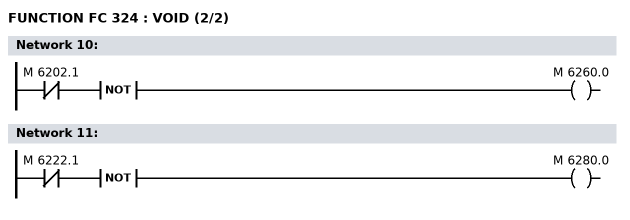

      AN    M   6202.1;
      NOT   ;
      =     M   6260.0;
NETWORK
TITLE =

      AN    M   6222.1;
      NOT   ;
      =     M   6280.0;
END_FUNCTION

FUNCTION_BLOCK FB 406
TITLE =Data Block Move Program
AUTHOR : HMC
FAMILY : Car_Type
NAME : Car_Type
VERSION : 1.0


VAR_INPUT
  FWD_Pulse : BOOL ;
  RET_Pulse : BOOL ;
  Source_DB : INT ;
  Start_Add : INT ;
  Stn_Amount : INT ;
  Byte_per_Stn : INT ;
  Cpu_Run_Pulse : BOOL ;
END_VAR
VAR_OUTPUT
  Complete : BOOL ;
END_VAR
VAR
  Operation : BOOL ;
  Mask_Arr : ARRAY  [0 .. 599 ] OF BYTE ;
  Ret : INT ;
  Data_Type : WORD ;
  Data_Length : INT ;
  Secend_Stn_Add : INT ;
  Fill_Source : WORD ;
END_VAR
VAR_TEMP
  First_Stn : ANY ;
  Mask : ANY ;
  Second_Stn : ANY ;
  Save_AR1 : DWORD ;
  Save_AR2 : DWORD ;
  Save_DB : INT ;
  Save_DI : INT ;
  First_Stn_1 : ANY ;
END_VAR
BEGIN
NETWORK
TITLE =Save adress register and DB's

      TAR1  #Save_AR1; // Save adress register 1
      TAR2  #Save_AR2; // Save adress register 2
      L     DBNO; // loads the number of the shared open data block
      T     #Save_DB;
      L     DINO; // loads the number of the opened instance data block
      T     #Save_DI;
NETWORK
TITLE =Operation Pulse

      O     #FWD_Pulse; // External ForwardOperation Signal
      O     #RET_Pulse; // External Return Operation Signal
      FP    #Operation; // Operation Pulse
      JNB   _End; // Jump to End
NETWORK
TITLE =Data Type Select In ANY Type Parameter

      A(    ; // If Source DB is Not Zero
      L     #Source_DB;
      L     0;
      <>I   ;
      )     ;
      JNB   _001; // Jump to Next Step
      L     W#16#8400; // Load "8400" _ Means "DB Area"
      T     #Data_Type; // Transfer to Data_Type
_001: NOP   0;
NETWORK
TITLE =Data Type Select In ANY Type Parameter

      A(    ; // If DB_NO is Zero
      L     #Source_DB;
      L     0;
      ==I   ;
      )     ;
      JNB   _002; // Jump to Next Step
      L     W#16#8300; // Load "8300" _ Means "Bit Memory Area"
      T     #Data_Type; // Transfer to Data_Type
_002: NOP   0;
NETWORK
TITLE =Data Length Select

      L     #Stn_Amount; // Station Amount - 1
      L     1;
      -I    ;
      L     #Byte_per_Stn; // Multi Length Per Station
      *I    ;
      T     #Data_Length; // Transfer to Data Length
NETWORK
TITLE =2nd Station Address Select

      L     #Start_Add; // Pluse Start Address And Length
      L     #Byte_per_Stn;
      +I    ;
      T     #Secend_Stn_Add; // Transfer to Second Station Address
NETWORK
TITLE =Make a "ANY" Type Data

      LAR1  P##First_Stn; // Load 1st Station Address of ANY Pointer In "AR1"

      L     B#16#10; // Load Syntax ID For S7 "10"
      T     LB [AR1,P#0.0]; // Transfer ID to the ANY Pointer

      L     B#16#2; // Load Data Type _ "2" means "BYTE"
      T     LB [AR1,P#1.0]; // Transfer Data Type to the ANY Pointer

      L     #Data_Length; // Load the Length of Source Data
      T     LW [AR1,P#2.0]; // Transfer the Numbers to the ANY Pointer

      L     #Source_DB; // Load DB Number _ "0" means don't use "DB"
      T     LW [AR1,P#4.0]; // Transfer the Numbers to the ANY Pointer

      L     #Data_Type; // Load Data Type _ "83" means "Bit Memory" Area
      T     LW [AR1,P#6.0]; //                  "84" means "DB" Area

      L     #Start_Add; // Load Start Address
      SLW   3; // Shift Left Word _ "3" Bit
      T     LW [AR1,P#8.0]; // Transfer the Address to the ANY Pointer

      LAR1  P##Mask; // Load 2nd Station Address of ANY Pointer In "AR1"

      L     B#16#10; //Load Syntax ID For S7 "10"
      T     LB [AR1,P#0.0]; //Load Syntax ID For S7 "10"

      L     B#16#2; //  Load Data Type _ "2" means "BYTE"
      T     LB [AR1,P#1.0]; // Transfer Data Type to the ANY Pointer

      L     #Data_Length; // Load the Length of Target Data
      T     LW [AR1,P#2.0]; // Transfer the Numbers to the ANY Pointer

      L     #Save_DI; // Load DB Number _ "0" means don't use "DB"
      T     LW [AR1,P#4.0]; // Transfer the Numbers to the ANY Pointer

      L     #Data_Type; // Load Data Type _ "83" means "Bit Memory" Area
      T     LW [AR1,P#6.0]; //                  "84" means "DB" Area

      L     16; //  Load Start Address
      SLW   3; // Shift Left Word _ "3" Bit
      T     LW [AR1,P#8.0]; // Transfer the Address to the ANY Pointer

NETWORK
TITLE =Make a "ANY" Type Data

      LAR1  P##Second_Stn; // Load 1st Station Address of ANY Pointer In "AR1"

      L     B#16#10; // Load Syntax ID For S7 "10"
      T     LB [AR1,P#0.0]; // Transfer ID to the ANY Pointer

      L     B#16#2; // Load Data Type _ "2" means "BYTE"
      T     LB [AR1,P#1.0]; // Transfer Data Type to the ANY Pointer

      L     #Data_Length; // Load the Length of Source Data
      T     LW [AR1,P#2.0]; // Transfer the Numbers to the ANY Pointer

      L     #Source_DB; // Load DB Number _ "0" means don't use "DB"
      T     LW [AR1,P#4.0]; // Transfer the Numbers to the ANY Pointer

      L     #Data_Type; // Load Data Type _ "83" means "Bit Memory" Area
      T     LW [AR1,P#6.0]; //                  "84" means "DB" Area

      L     #Secend_Stn_Add; // Load Second Station Address
      SLW   3; // Shift Left Word _ "3" Bit
      T     LW [AR1,P#8.0]; // Transfer the Address to the ANY Pointer
NETWORK
TITLE =Reset Car Type Transfer Complete Signal

      O     #FWD_Pulse; // External Forward Operation Signal
      O     #RET_Pulse; // External Return Operation Signal
      R     #Complete; // Reset Complete Signal
NETWORK
TITLE =Make Fill Source Data

      L     0;
      T     #Fill_Source;
NETWORK
TITLE =Fwd Block Move to Mask Area

      A     #FWD_Pulse; // External Forward Operation Signal
      AN    #Complete; // Complete Signal is False
      AN    #Cpu_Run_Pulse;
      JNB   _FWD;
      CALL SFC   20 (
           SRCBLK                   := #First_Stn,
           RET_VAL                  := #Ret,
           DSTBLK                   := #Mask);

NETWORK
TITLE =Clear Source Data Area


      CALL SFC   21 (
           BVAL                     := #Fill_Source,// "Zero"
           RET_VAL                  := #Ret,
           BLK                      := #First_Stn);// Transfer to First Station Area

NETWORK
TITLE =Fwd Block Move to Second Station Area


      CALL SFC   20 (
           SRCBLK                   := #Mask,
           RET_VAL                  := #Ret,
           DSTBLK                   := #Second_Stn);

NETWORK
TITLE =Clear Mask Data Area


      CALL SFC   21 (
           BVAL                     := #Fill_Source,// "Zero"
           RET_VAL                  := #Ret,
           BLK                      := #Mask);// Transfer to Mask Area
_FWD: NOP   0;
NETWORK
TITLE =Rev Block Move to Mask Area

      A     #RET_Pulse; // External Return Operation Signal
      AN    #Complete; // Complete Signal is False
      AN    #Cpu_Run_Pulse;
      JNB   _REV;
      CALL SFC   20 (
           SRCBLK                   := #Second_Stn,
           RET_VAL                  := #Ret,
           DSTBLK                   := #Mask);

NETWORK
TITLE =Clear Source Data Area


      CALL SFC   21 (
           BVAL                     := #Fill_Source,// "Zero"
           RET_VAL                  := #Ret,
           BLK                      := #Second_Stn);// Transfer to Second Station Area

NETWORK
TITLE =Rev Block Move to First Station Area


      CALL SFC   20 (
           SRCBLK                   := #Mask,
           RET_VAL                  := #Ret,
           DSTBLK                   := #First_Stn);

NETWORK
TITLE =Clear Mask Data Area


      CALL SFC   21 (
           BVAL                     := #Fill_Source,// "Zero"
           RET_VAL                  := #Ret,
           BLK                      := #Mask);// Transfer to Mask Area
_REV: NOP   0;
NETWORK
TITLE =Set Complete Signal

      S     #Complete;
_End: NOP   0;
END_FUNCTION_BLOCK

FUNCTION_BLOCK FB 426
TITLE =Sensor Error,Lamp Variables Program
AUTHOR : HMC
FAMILY : Common
NAME : Common
VERSION : 1.0


VAR_INPUT
  Enable_Aux : BOOL ;
  Adv_Amount : INT ;
  Ret_Amount : INT ;
  LS_Adv1 : BOOL ;
  LS_Ret1 : BOOL ;
  LS_Adv2 : BOOL ;
  LS_Ret2 : BOOL ;
  LS_Adv3 : BOOL ;
  LS_Ret3 : BOOL ;
  LS_Adv4 : BOOL ;
  LS_Ret4 : BOOL ;
  LS_Adv5 : BOOL ;
  LS_Ret5 : BOOL ;
  LS_Adv6 : BOOL ;
  LS_Ret6 : BOOL ;
  LS_Adv7 : BOOL ;
  LS_Ret7 : BOOL ;
  LS_Adv8 : BOOL ;
  LS_Ret8 : BOOL ;
  SOL_Adv : BOOL ;
  SOL_Ret : BOOL ;
  M_Ready : BOOL ;
  T_CHK1 : TIME ;
  T_CHK2 : TIME ;
  PB_Lamp_CHK : BOOL ;
  PB_Error_Rst : BOOL ;
  M_FLICK : BOOL ;
END_VAR
VAR_OUTPUT
  M_Adv_Err : BOOL ;
  M_Ret_Err : BOOL ;
  LP_Adv : BOOL ;
  LP_Ret : BOOL ;
  Visu_Adv : WORD ;
  Visu_Ret : WORD ;
END_VAR
VAR
  Error_T1 : SFB 4;
  Error_T2 : SFB 4;
  Adv_End_Aux : BOOL ;
  Ret_End_Aux : BOOL ;
  CHK_Aux1 : BOOL ;
  CHK_Aux2 : BOOL ;
  Error_T1_DN : BOOL ;
  Error_T2_DN : BOOL ;
  Adv_Memo : BOOL ;
  Visu_Adv_Arr : ARRAY  [0 .. 15 ] OF BOOL ;
  Visu_Ret_Arr : ARRAY  [0 .. 15 ] OF BOOL ;
  BLK_Move_Ret : INT ;
  Enable : BOOL ;
  Adv_End : BOOL ;
  Ret_End : BOOL ;
END_VAR
BEGIN
NETWORK
TITLE =
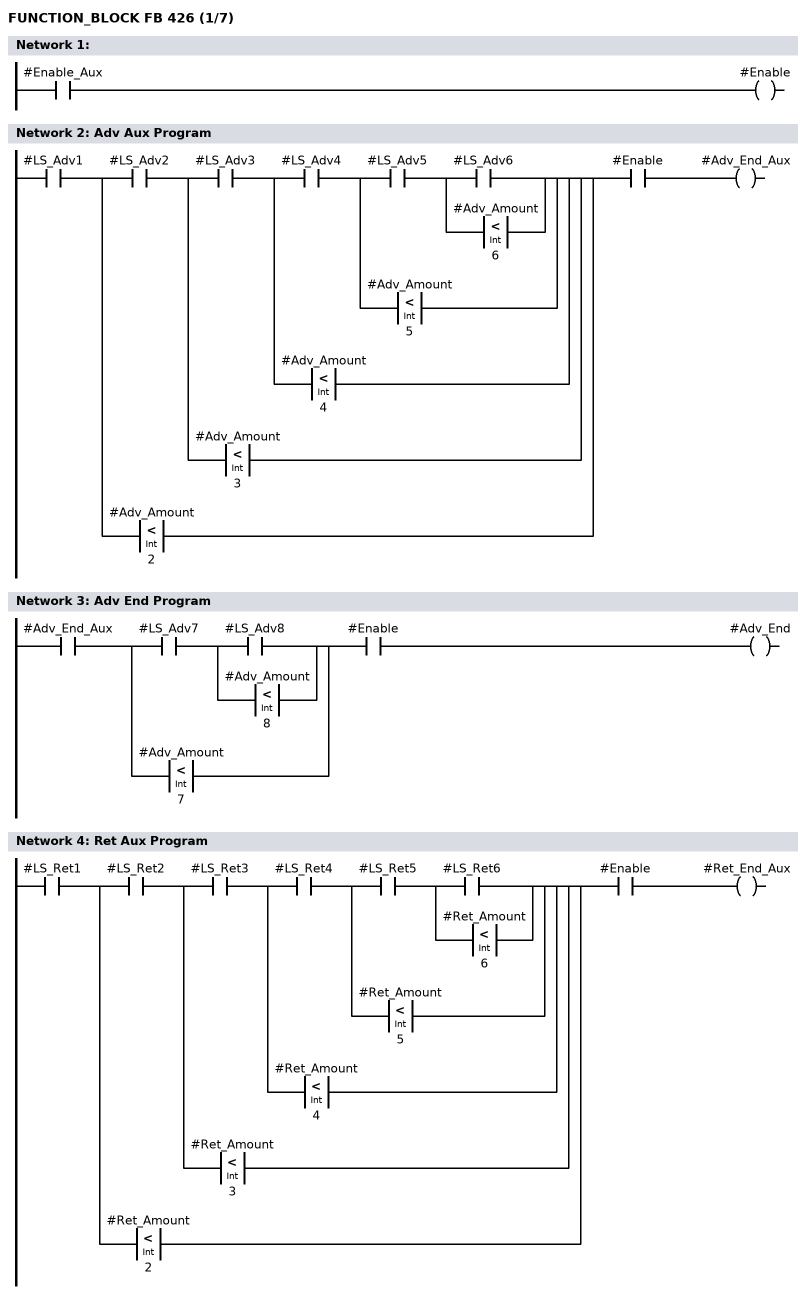

      A     #Enable_Aux;
      =     #Enable;
NETWORK
TITLE =Adv Aux Program

      A     #LS_Adv1;
      A(    ;
      A     #LS_Adv2;
      A(    ;
      A     #LS_Adv3;
      A(    ;
      A     #LS_Adv4;
      A(    ;
      A     #LS_Adv5;
      A(    ;
      O     #LS_Adv6;
      O(    ;
      L     #Adv_Amount;
      L     6;
      <I    ;
      )     ;
      )     ;
      O(    ;
      L     #Adv_Amount;
      L     5;
      <I    ;
      )     ;
      )     ;
      O(    ;
      L     #Adv_Amount;
      L     4;
      <I    ;
      )     ;
      )     ;
      O(    ;
      L     #Adv_Amount;
      L     3;
      <I    ;
      )     ;
      )     ;
      O(    ;
      L     #Adv_Amount;
      L     2;
      <I    ;
      )     ;
      )     ;
      A     #Enable;
      =     #Adv_End_Aux;
NETWORK
TITLE =Adv End Program

      A     #Adv_End_Aux;
      A(    ;
      A     #LS_Adv7;
      A(    ;
      O     #LS_Adv8;
      O(    ;
      L     #Adv_Amount;
      L     8;
      <I    ;
      )     ;
      )     ;
      O(    ;
      L     #Adv_Amount;
      L     7;
      <I    ;
      )     ;
      )     ;
      A     #Enable;
      =     #Adv_End;
NETWORK
TITLE =Ret Aux Program

      A     #LS_Ret1;
      A(    ;
      A     #LS_Ret2;
      A(    ;
      A     #LS_Ret3;
      A(    ;
      A     #LS_Ret4;
      A(    ;
      A     #LS_Ret5;
      A(    ;
      O     #LS_Ret6;
      O(    ;
      L     #Ret_Amount;
      L     6;
      <I    ;
      )     ;
      )     ;
      O(    ;
      L     #Ret_Amount;
      L     5;
      <I    ;
      )     ;
      )     ;
      O(    ;
      L     #Ret_Amount;
      L     4;
      <I    ;
      )     ;
      )     ;
      O(    ;
      L     #Ret_Amount;
      L     3;
      <I    ;
      )     ;
      )     ;
      O(    ;
      L     #Ret_Amount;
      L     2;
      <I    ;
      )     ;
      )     ;
      A     #Enable;
      =     #Ret_End_Aux;
NETWORK
TITLE =Ret End Program
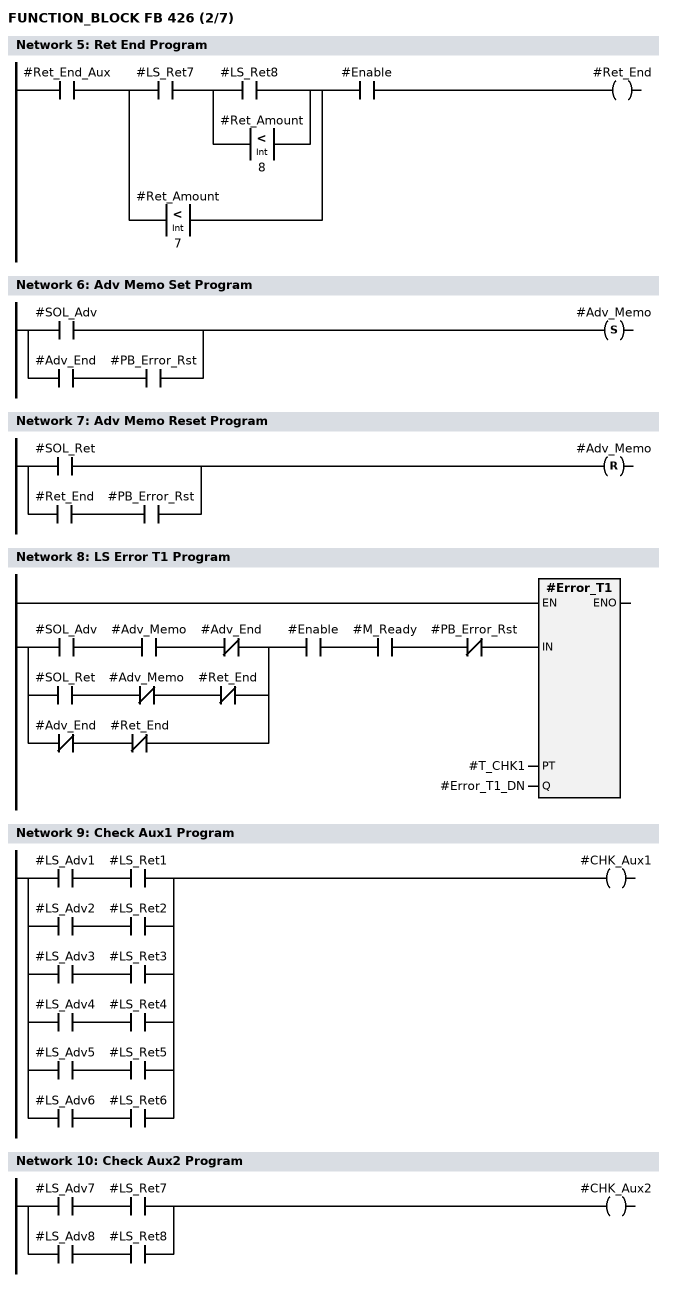

      A     #Ret_End_Aux;
      A(    ;
      A     #LS_Ret7;
      A(    ;
      O     #LS_Ret8;
      O(    ;
      L     #Ret_Amount;
      L     8;
      <I    ;
      )     ;
      )     ;
      O(    ;
      L     #Ret_Amount;
      L     7;
      <I    ;
      )     ;
      )     ;
      A     #Enable;
      =     #Ret_End;
NETWORK
TITLE =Adv Memo Set Program

      O     #SOL_Adv;
      O     ;
      A     #Adv_End;
      A     #PB_Error_Rst;
      S     #Adv_Memo;
NETWORK
TITLE =Adv Memo Reset Program

      O     #SOL_Ret;
      O     ;
      A     #Ret_End;
      A     #PB_Error_Rst;
      R     #Adv_Memo;
NETWORK
TITLE =LS Error T1 Program

      A(    ;
      A     #SOL_Adv;
      A     #Adv_Memo;
      AN    #Adv_End;
      O     ;
      A     #SOL_Ret;
      AN    #Adv_Memo;
      AN    #Ret_End;
      O     ;
      AN    #Adv_End;
      AN    #Ret_End;
      )     ;
      A     #Enable;
      A     #M_Ready;
      AN    #PB_Error_Rst;
      =     L      0.0;
      BLD   103;
      CALL #Error_T1 (
           IN                       := L      0.0,
           PT                       := #T_CHK1,
           Q                        := #Error_T1_DN);

      NOP   0;
NETWORK
TITLE =Check Aux1 Program

      A     #LS_Adv1;
      A     #LS_Ret1;
      O     ;
      A     #LS_Adv2;
      A     #LS_Ret2;
      O     ;
      A     #LS_Adv3;
      A     #LS_Ret3;
      O     ;
      A     #LS_Adv4;
      A     #LS_Ret4;
      O     ;
      A     #LS_Adv5;
      A     #LS_Ret5;
      O     ;
      A     #LS_Adv6;
      A     #LS_Ret6;
      =     #CHK_Aux1;
NETWORK
TITLE =Check Aux2 Program

      A     #LS_Adv7;
      A     #LS_Ret7;
      O     ;
      A     #LS_Adv8;
      A     #LS_Ret8;
      =     #CHK_Aux2;
NETWORK
TITLE =LS Error T2 Program
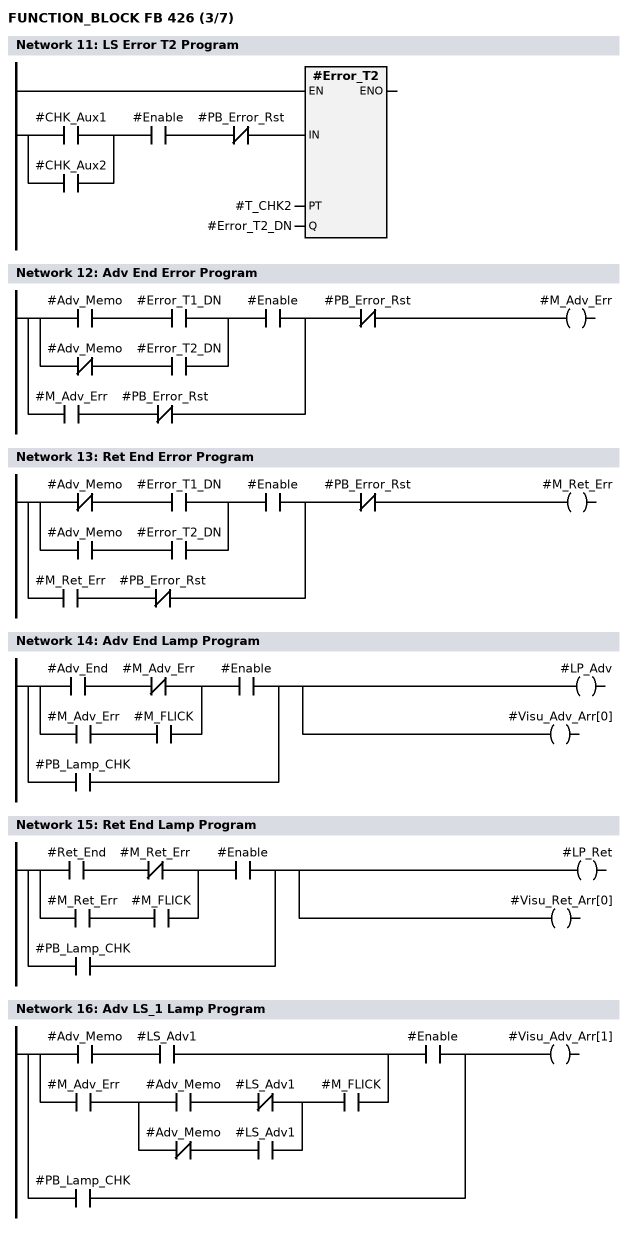

      A(    ;
      O     #CHK_Aux1;
      O     #CHK_Aux2;
      )     ;
      A     #Enable;
      AN    #PB_Error_Rst;
      =     L      0.0;
      BLD   103;
      CALL #Error_T2 (
           IN                       := L      0.0,
           PT                       := #T_CHK2,
           Q                        := #Error_T2_DN);

      NOP   0;
NETWORK
TITLE =Adv End Error Program

      A(    ;
      A(    ;
      A     #Adv_Memo;
      A     #Error_T1_DN;
      O     ;
      AN    #Adv_Memo;
      A     #Error_T2_DN;
      )     ;
      A     #Enable;
      O     ;
      A     #M_Adv_Err;
      AN    #PB_Error_Rst;
      )     ;
      AN    #PB_Error_Rst;
      =     #M_Adv_Err;
NETWORK
TITLE =Ret End Error Program

      A(    ;
      A(    ;
      AN    #Adv_Memo;
      A     #Error_T1_DN;
      O     ;
      A     #Adv_Memo;
      A     #Error_T2_DN;
      )     ;
      A     #Enable;
      O     ;
      A     #M_Ret_Err;
      AN    #PB_Error_Rst;
      )     ;
      AN    #PB_Error_Rst;
      =     #M_Ret_Err;
NETWORK
TITLE =Adv End Lamp Program

      A(    ;
      A     #Adv_End;
      AN    #M_Adv_Err;
      O     ;
      A     #M_Adv_Err;
      A     #M_FLICK;
      )     ;
      A     #Enable;
      O     #PB_Lamp_CHK;
      =     #LP_Adv;
      =     #Visu_Adv_Arr[0];
NETWORK
TITLE =Ret End Lamp Program

      A(    ;
      A     #Ret_End;
      AN    #M_Ret_Err;
      O     ;
      A     #M_Ret_Err;
      A     #M_FLICK;
      )     ;
      A     #Enable;
      O     #PB_Lamp_CHK;
      =     #LP_Ret;
      =     #Visu_Ret_Arr[0];
NETWORK
TITLE =Adv LS_1 Lamp Program

      A(    ;
      A     #Adv_Memo;
      A     #LS_Adv1;
      O     ;
      A     #M_Adv_Err;
      A(    ;
      A     #Adv_Memo;
      AN    #LS_Adv1;
      O     ;
      AN    #Adv_Memo;
      A     #LS_Adv1;
      )     ;
      A     #M_FLICK;
      )     ;
      A     #Enable;
      O     #PB_Lamp_CHK;
      =     #Visu_Adv_Arr[1];
NETWORK
TITLE =Adv LS_2 Lamp Program
//
//
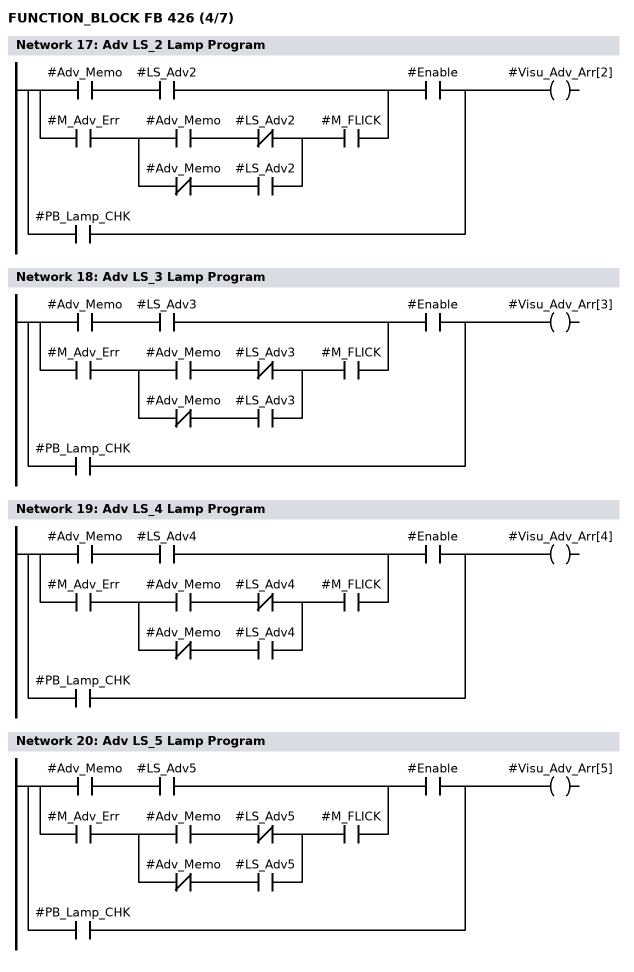
      A(    ;
      A     #Adv_Memo;
      A     #LS_Adv2;
      O     ;
      A     #M_Adv_Err;
      A(    ;
      A     #Adv_Memo;
      AN    #LS_Adv2;
      O     ;
      AN    #Adv_Memo;
      A     #LS_Adv2;
      )     ;
      A     #M_FLICK;
      )     ;
      A     #Enable;
      O     #PB_Lamp_CHK;
      =     #Visu_Adv_Arr[2];
NETWORK
TITLE =Adv LS_3 Lamp Program
//
//
      A(    ;
      A     #Adv_Memo;
      A     #LS_Adv3;
      O     ;
      A     #M_Adv_Err;
      A(    ;
      A     #Adv_Memo;
      AN    #LS_Adv3;
      O     ;
      AN    #Adv_Memo;
      A     #LS_Adv3;
      )     ;
      A     #M_FLICK;
      )     ;
      A     #Enable;
      O     #PB_Lamp_CHK;
      =     #Visu_Adv_Arr[3];
NETWORK
TITLE =Adv LS_4 Lamp Program
//
//
      A(    ;
      A     #Adv_Memo;
      A     #LS_Adv4;
      O     ;
      A     #M_Adv_Err;
      A(    ;
      A     #Adv_Memo;
      AN    #LS_Adv4;
      O     ;
      AN    #Adv_Memo;
      A     #LS_Adv4;
      )     ;
      A     #M_FLICK;
      )     ;
      A     #Enable;
      O     #PB_Lamp_CHK;
      =     #Visu_Adv_Arr[4];
NETWORK
TITLE =Adv LS_5 Lamp Program
//
//
      A(    ;
      A     #Adv_Memo;
      A     #LS_Adv5;
      O     ;
      A     #M_Adv_Err;
      A(    ;
      A     #Adv_Memo;
      AN    #LS_Adv5;
      O     ;
      AN    #Adv_Memo;
      A     #LS_Adv5;
      )     ;
      A     #M_FLICK;
      )     ;
      A     #Enable;
      O     #PB_Lamp_CHK;
      =     #Visu_Adv_Arr[5];
NETWORK
TITLE =Adv LS_6 Lamp Program
//
//
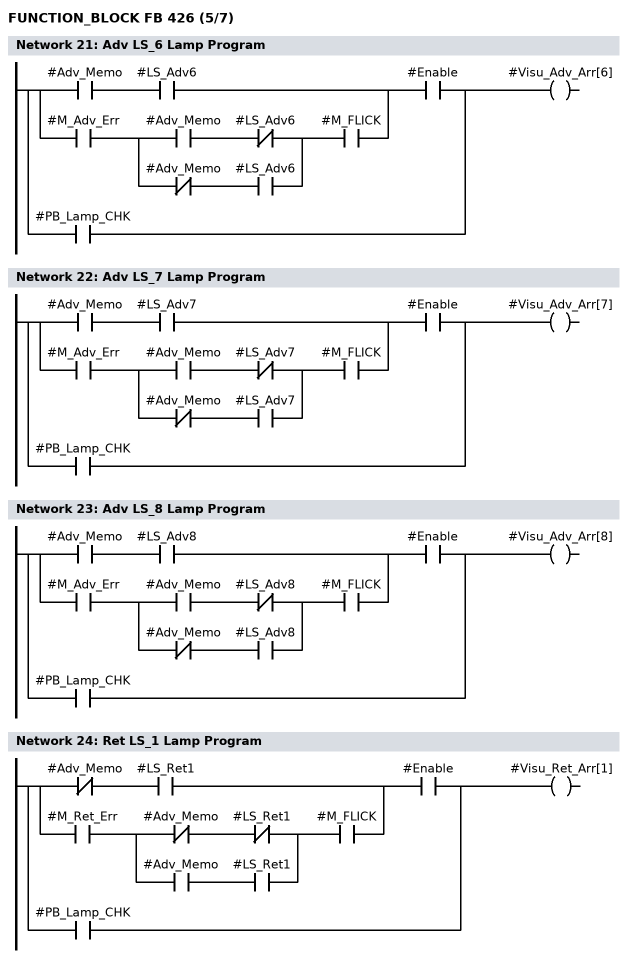
      A(    ;
      A     #Adv_Memo;
      A     #LS_Adv6;
      O     ;
      A     #M_Adv_Err;
      A(    ;
      A     #Adv_Memo;
      AN    #LS_Adv6;
      O     ;
      AN    #Adv_Memo;
      A     #LS_Adv6;
      )     ;
      A     #M_FLICK;
      )     ;
      A     #Enable;
      O     #PB_Lamp_CHK;
      =     #Visu_Adv_Arr[6];
NETWORK
TITLE =Adv LS_7 Lamp Program
//
//
      A(    ;
      A     #Adv_Memo;
      A     #LS_Adv7;
      O     ;
      A     #M_Adv_Err;
      A(    ;
      A     #Adv_Memo;
      AN    #LS_Adv7;
      O     ;
      AN    #Adv_Memo;
      A     #LS_Adv7;
      )     ;
      A     #M_FLICK;
      )     ;
      A     #Enable;
      O     #PB_Lamp_CHK;
      =     #Visu_Adv_Arr[7];
NETWORK
TITLE =Adv LS_8 Lamp Program
//
//
      A(    ;
      A     #Adv_Memo;
      A     #LS_Adv8;
      O     ;
      A     #M_Adv_Err;
      A(    ;
      A     #Adv_Memo;
      AN    #LS_Adv8;
      O     ;
      AN    #Adv_Memo;
      A     #LS_Adv8;
      )     ;
      A     #M_FLICK;
      )     ;
      A     #Enable;
      O     #PB_Lamp_CHK;
      =     #Visu_Adv_Arr[8];
NETWORK
TITLE =Ret LS_1 Lamp Program
//
//
      A(    ;
      AN    #Adv_Memo;
      A     #LS_Ret1;
      O     ;
      A     #M_Ret_Err;
      A(    ;
      AN    #Adv_Memo;
      AN    #LS_Ret1;
      O     ;
      A     #Adv_Memo;
      A     #LS_Ret1;
      )     ;
      A     #M_FLICK;
      )     ;
      A     #Enable;
      O     #PB_Lamp_CHK;
      =     #Visu_Ret_Arr[1];
NETWORK
TITLE =Ret LS_2 Lamp Program
//
//
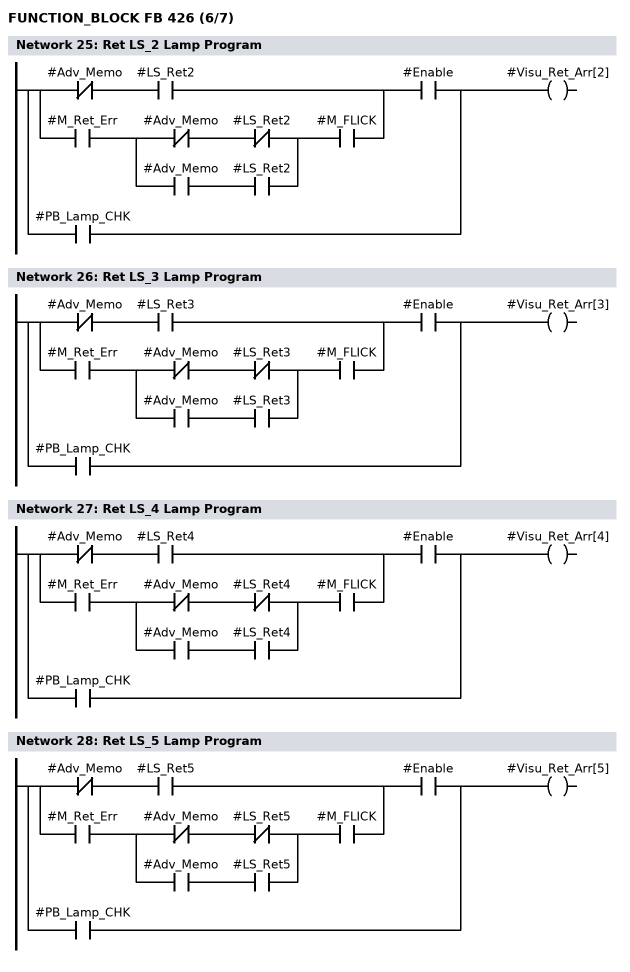
      A(    ;
      AN    #Adv_Memo;
      A     #LS_Ret2;
      O     ;
      A     #M_Ret_Err;
      A(    ;
      AN    #Adv_Memo;
      AN    #LS_Ret2;
      O     ;
      A     #Adv_Memo;
      A     #LS_Ret2;
      )     ;
      A     #M_FLICK;
      )     ;
      A     #Enable;
      O     #PB_Lamp_CHK;
      =     #Visu_Ret_Arr[2];
NETWORK
TITLE =Ret LS_3 Lamp Program
//
//
      A(    ;
      AN    #Adv_Memo;
      A     #LS_Ret3;
      O     ;
      A     #M_Ret_Err;
      A(    ;
      AN    #Adv_Memo;
      AN    #LS_Ret3;
      O     ;
      A     #Adv_Memo;
      A     #LS_Ret3;
      )     ;
      A     #M_FLICK;
      )     ;
      A     #Enable;
      O     #PB_Lamp_CHK;
      =     #Visu_Ret_Arr[3];
NETWORK
TITLE =Ret LS_4 Lamp Program
//
//
      A(    ;
      AN    #Adv_Memo;
      A     #LS_Ret4;
      O     ;
      A     #M_Ret_Err;
      A(    ;
      AN    #Adv_Memo;
      AN    #LS_Ret4;
      O     ;
      A     #Adv_Memo;
      A     #LS_Ret4;
      )     ;
      A     #M_FLICK;
      )     ;
      A     #Enable;
      O     #PB_Lamp_CHK;
      =     #Visu_Ret_Arr[4];
NETWORK
TITLE =Ret LS_5 Lamp Program
//
//
      A(    ;
      AN    #Adv_Memo;
      A     #LS_Ret5;
      O     ;
      A     #M_Ret_Err;
      A(    ;
      AN    #Adv_Memo;
      AN    #LS_Ret5;
      O     ;
      A     #Adv_Memo;
      A     #LS_Ret5;
      )     ;
      A     #M_FLICK;
      )     ;
      A     #Enable;
      O     #PB_Lamp_CHK;
      =     #Visu_Ret_Arr[5];
NETWORK
TITLE =Ret LS_6 Lamp Program
//
//
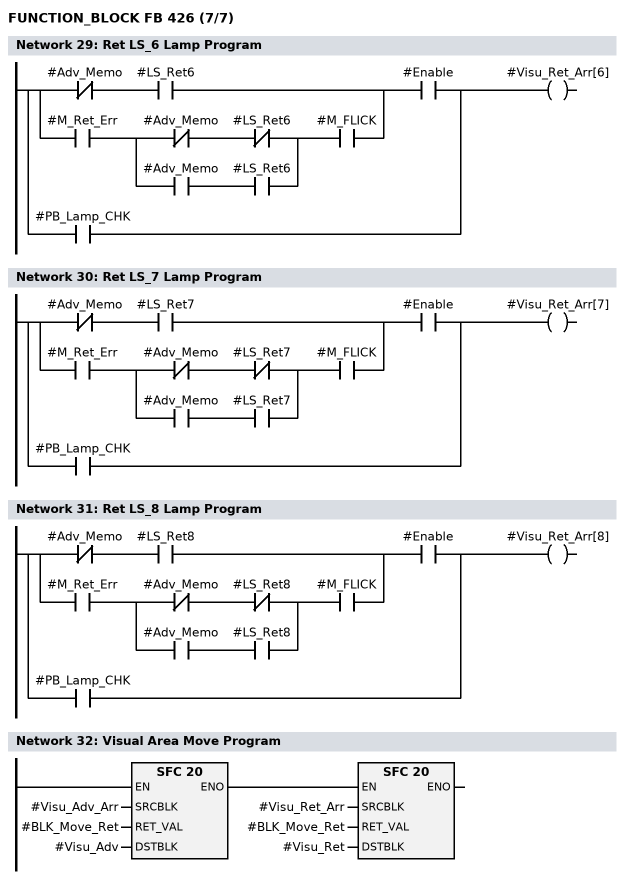
      A(    ;
      AN    #Adv_Memo;
      A     #LS_Ret6;
      O     ;
      A     #M_Ret_Err;
      A(    ;
      AN    #Adv_Memo;
      AN    #LS_Ret6;
      O     ;
      A     #Adv_Memo;
      A     #LS_Ret6;
      )     ;
      A     #M_FLICK;
      )     ;
      A     #Enable;
      O     #PB_Lamp_CHK;
      =     #Visu_Ret_Arr[6];
NETWORK
TITLE =Ret LS_7 Lamp Program
//
//
      A(    ;
      AN    #Adv_Memo;
      A     #LS_Ret7;
      O     ;
      A     #M_Ret_Err;
      A(    ;
      AN    #Adv_Memo;
      AN    #LS_Ret7;
      O     ;
      A     #Adv_Memo;
      A     #LS_Ret7;
      )     ;
      A     #M_FLICK;
      )     ;
      A     #Enable;
      O     #PB_Lamp_CHK;
      =     #Visu_Ret_Arr[7];
NETWORK
TITLE =Ret LS_8 Lamp Program
//
//
      A(    ;
      AN    #Adv_Memo;
      A     #LS_Ret8;
      O     ;
      A     #M_Ret_Err;
      A(    ;
      AN    #Adv_Memo;
      AN    #LS_Ret8;
      O     ;
      A     #Adv_Memo;
      A     #LS_Ret8;
      )     ;
      A     #M_FLICK;
      )     ;
      A     #Enable;
      O     #PB_Lamp_CHK;
      =     #Visu_Ret_Arr[8];
NETWORK
TITLE =Visual Area Move Program

      A(    ;
      CALL SFC   20 (
           SRCBLK                   := #Visu_Adv_Arr,
           RET_VAL                  := #BLK_Move_Ret,
           DSTBLK                   := #Visu_Adv);
      A     BR;
      )     ;
      JNB   _001;
      CALL SFC   20 (
           SRCBLK                   := #Visu_Ret_Arr,
           RET_VAL                  := #BLK_Move_Ret,
           DSTBLK                   := #Visu_Ret);
_001: NOP   0;
END_FUNCTION_BLOCK

FUNCTION_BLOCK FB 475
TITLE =ProfiBus DP Communication Fault Variables Program
AUTHOR : HMC
FAMILY : Drive
NAME : Drive
VERSION : 1.0


VAR_INPUT
  M_Check_Active : BOOL ;
  DP_Not_Pre_Byte : BYTE ;	//Startadress Outputs from HW-Konfig
  DP_Error_Byte : BYTE ;	//Startadress Inputs from HW-Konfig
  M_Error_Rst : BOOL ;
END_VAR
VAR_OUTPUT
  Node0_Fault : BOOL ;
  Node1_Fault : BOOL ;
  Node2_Fault : BOOL ;
  Node3_Fault : BOOL ;
  Node4_Fault : BOOL ;
  Node5_Fault : BOOL ;
  Node6_Fault : BOOL ;
  Node7_Fault : BOOL ;
END_VAR
VAR
  Pre_Arr : ARRAY  [0 .. 7 ] OF BOOL ;
  Fault_Arr : ARRAY  [0 .. 7 ] OF BOOL ;
  node_0_err : SFB 4;
  node_1_err : SFB 4;
  node_2_err : SFB 4;
  node_3_err : SFB 4;
  node_4_err : SFB 4;
  node_5_err : SFB 4;
  node_6_err : SFB 4;
  node_7_err : SFB 4;
END_VAR
VAR_TEMP
  Ret : INT ;
END_VAR
BEGIN
NETWORK
TITLE =DP Fault Byte Move To DP Fault Array
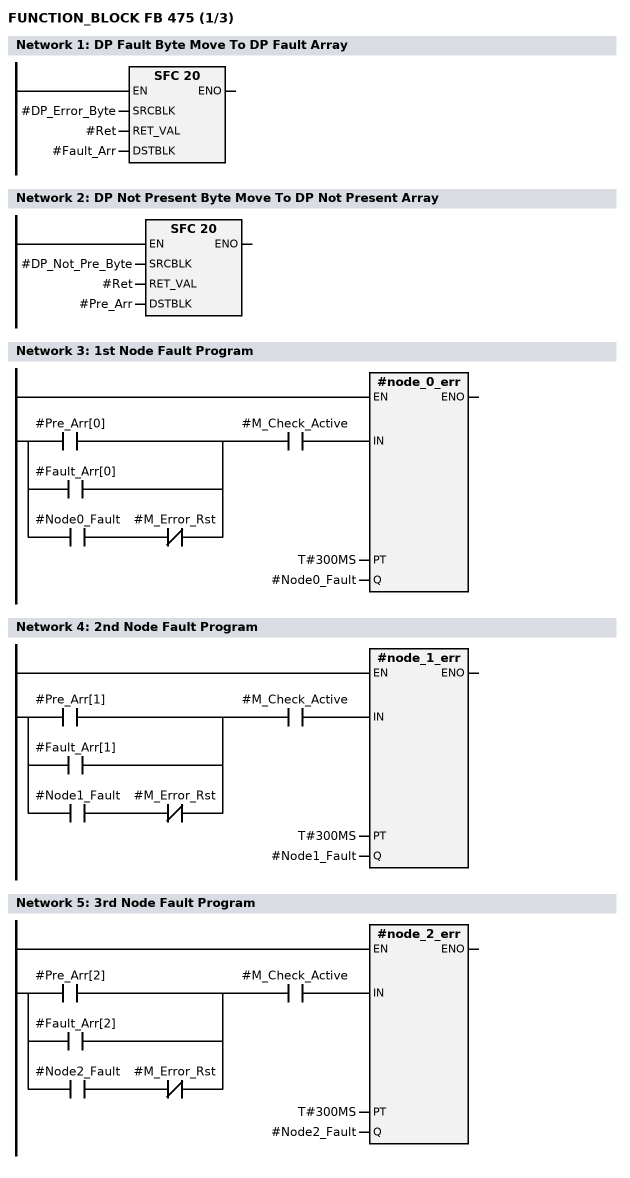

      CALL SFC   20 (
           SRCBLK                   := #DP_Error_Byte,
           RET_VAL                  := #Ret,
           DSTBLK                   := #Fault_Arr);
      NOP   0;
NETWORK
TITLE =DP Not Present Byte Move To DP Not Present Array

      CALL SFC   20 (
           SRCBLK                   := #DP_Not_Pre_Byte,
           RET_VAL                  := #Ret,
           DSTBLK                   := #Pre_Arr);
      NOP   0;
NETWORK
TITLE =1st Node Fault Program

      A(    ;
      O     #Pre_Arr[0];
      O     #Fault_Arr[0];
      O     ;
      A     #Node0_Fault;
      AN    #M_Error_Rst;
      )     ;
      A     #M_Check_Active;
      =     L      2.0;
      BLD   103;
      CALL #node_0_err (
           IN                       := L      2.0,
           PT                       := T#300MS,
           Q                        := #Node0_Fault);

      NOP   0;
NETWORK
TITLE =2nd Node Fault Program

      A(    ;
      O     #Pre_Arr[1];
      O     #Fault_Arr[1];
      O     ;
      A     #Node1_Fault;
      AN    #M_Error_Rst;
      )     ;
      A     #M_Check_Active;
      =     L      2.0;
      BLD   103;
      CALL #node_1_err (
           IN                       := L      2.0,
           PT                       := T#300MS,
           Q                        := #Node1_Fault);

      NOP   0;
NETWORK
TITLE =3rd Node Fault Program

      A(    ;
      O     #Pre_Arr[2];
      O     #Fault_Arr[2];
      O     ;
      A     #Node2_Fault;
      AN    #M_Error_Rst;
      )     ;
      A     #M_Check_Active;
      =     L      2.0;
      BLD   103;
      CALL #node_2_err (
           IN                       := L      2.0,
           PT                       := T#300MS,
           Q                        := #Node2_Fault);

      NOP   0;
NETWORK
TITLE =4th Node Fault Program
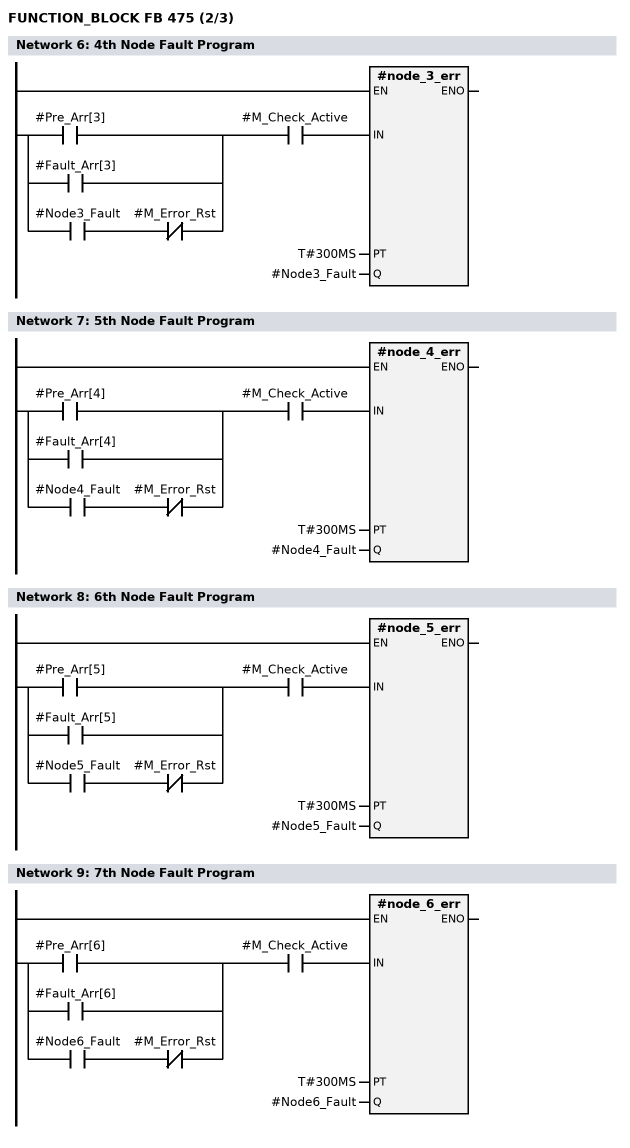

      A(    ;
      O     #Pre_Arr[3];
      O     #Fault_Arr[3];
      O     ;
      A     #Node3_Fault;
      AN    #M_Error_Rst;
      )     ;
      A     #M_Check_Active;
      =     L      2.0;
      BLD   103;
      CALL #node_3_err (
           IN                       := L      2.0,
           PT                       := T#300MS,
           Q                        := #Node3_Fault);

      NOP   0;
NETWORK
TITLE =5th Node Fault Program

      A(    ;
      O     #Pre_Arr[4];
      O     #Fault_Arr[4];
      O     ;
      A     #Node4_Fault;
      AN    #M_Error_Rst;
      )     ;
      A     #M_Check_Active;
      =     L      2.0;
      BLD   103;
      CALL #node_4_err (
           IN                       := L      2.0,
           PT                       := T#300MS,
           Q                        := #Node4_Fault);

      NOP   0;
NETWORK
TITLE =6th Node Fault Program

      A(    ;
      O     #Pre_Arr[5];
      O     #Fault_Arr[5];
      O     ;
      A     #Node5_Fault;
      AN    #M_Error_Rst;
      )     ;
      A     #M_Check_Active;
      =     L      2.0;
      BLD   103;
      CALL #node_5_err (
           IN                       := L      2.0,
           PT                       := T#300MS,
           Q                        := #Node5_Fault);

      NOP   0;
NETWORK
TITLE =7th Node Fault Program

      A(    ;
      O     #Pre_Arr[6];
      O     #Fault_Arr[6];
      O     ;
      A     #Node6_Fault;
      AN    #M_Error_Rst;
      )     ;
      A     #M_Check_Active;
      =     L      2.0;
      BLD   103;
      CALL #node_6_err (
           IN                       := L      2.0,
           PT                       := T#300MS,
           Q                        := #Node6_Fault);

      NOP   0;
NETWORK
TITLE =8th Node Fault Program
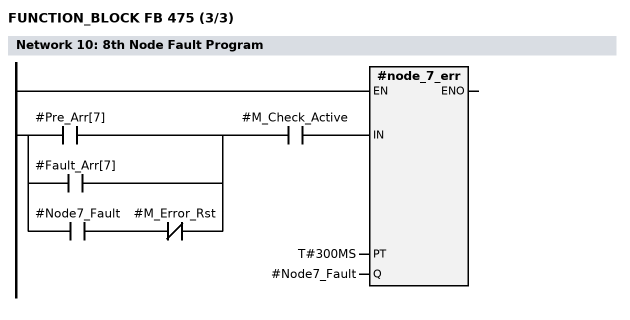

      A(    ;
      O     #Pre_Arr[7];
      O     #Fault_Arr[7];
      O     ;
      A     #Node7_Fault;
      AN    #M_Error_Rst;
      )     ;
      A     #M_Check_Active;
      =     L      2.0;
      BLD   103;
      CALL #node_7_err (
           IN                       := L      2.0,
           PT                       := T#300MS,
           Q                        := #Node7_Fault);

      NOP   0;
END_FUNCTION_BLOCK

FUNCTION FC 501 : VOID
TITLE =
VERSION : 0.1


VAR_INPUT
  FAC_No : INT ;	//Terminal No. 입력용
  FAC_DB_NO : INT ;	//생산지시용 DB 번호 입력용
  FAC_LOG_DB_NO : INT ;	//Terminal별 Log Data저장 DB 번호 입력용
  Line_Present_Data_DB_No : INT ;	//라인의 현재 공정 차종 영역이 저장된 DB번호 입력용
  Line_Present_Data_Byte : INT ;	//라인의 현재 공정 차종 영역이 저장된 DB의 Byte번호 입력용
  Order_Data_Send_DB_No : INT ;	//라인의 현재 공정에 서열 데이터를 수신할 DB번호 입력용
  Order_Data_Send_DB_Byte : INT ;	//라인의 현재 공정에 서열 데이터를 수신할 DB의 Byte번호 입력용
  ONLINE_Mode_Select : BOOL ;	//생산지시 ON/OFF 선택 스위치 또는 BIT 입력용
  Work_Complete : BOOL ;	//해당 공정의 작업완료 BIT 입력용
  Data_Shift_Condition : BOOL ;	//해당 공정에서 다음 공정으로 차종이 전송 되는 신호
  Data_Request : BOOL ;	//해당 공정에서 차종을 요구하는 신호
  BType_Change_Set_Rst_PB : BOOL ;	//수동으로 차종 Set/Reset 버튼
  Flicker_1s : BOOL ;	//PLC CPU에 정의된 1초 Clock용 신호
END_VAR
VAR_OUTPUT
  Communication_Error : BOOL ;	//terminal과 PLC간 통신 이상이 발생한 경우 출력
  Data_Error : BOOL ;	//Terminal에서 수신된 데이터에 이상이 발생한 경우 출력
END_VAR
VAR_TEMP
  Terminal : INT ;	//Terminal No. 저장 temp
  FAC_DB : INT ;	//생산지시용 DB 번호 저장 temp
  FAC_LOG_DB : INT ;	//Terminal별 Log Data저장 DB 번호 저장 temp
  LINE_PRESENT_DATA_DB : INT ;	//라인의 현재 공정 차종 영역이 저장된 DB번호 저장 temp
  ORDER_DATA_SEND_DB : INT ;	//라인의 현재 공정에 서열 데이터를 수신할 DB번호 저장 temp
  FAC_DB_Start_Byte_temp : INT ;	//Terminal별 FAC_DB의 시작 Byte 저장용
  FAC_DB_Start_Byte : INT ;	//Terminal별 FAC_DB의 시작 Byte 저장용
  NORMAL_ON : BOOL ;	//항상ON
  Present_RCV_VIN4 : WORD ;	//현재 수신된 데이터의 VIN No. 4자리
  Present_STA_VIN4 : WORD ;	//현재 공정 데이터의 VIN No. 4자리
  FAC_Data_NewValue : INT ;	//차종 설정 요청 정보의 데이터 변경 확인용 Temp1
  Final_Send_VIN : WORD ;	//차종 설정 요청 정보의 데이터 변경 확인용 Temp2
  Data_SET_Req_Count : INT ;	//차종 설정 요청 신호 발생 횟수 Temp
  Fill_start_point : INT ;
  BLKMove_Sourcstart_point : INT ;
  BLKMove_Deststart_point : INT ;
END_VAR
BEGIN
NETWORK
TITLE =FAC용 DB OPEN

      L     #FAC_No; //Terminal번호 Load
      T     #Terminal; //Terminal번호 Temp영역에 저장
      L     #FAC_DB_NO; //생산지시용 FAC DB번호 Load
      T     #FAC_DB; //생산지시용 FAC DB번호 Temp영역에 저장
      L     #FAC_LOG_DB_NO; //FAC Log 저장 DB번호 Load
      T     #FAC_LOG_DB; //FAC Log 저장 DB번호 Temp영역에 저장
      L     #Line_Present_Data_DB_No; //라인의 현재 공정 차종 영역이 저장된 DB번호 Load
      T     #LINE_PRESENT_DATA_DB; //라인의 현재 공정 차종 영역이 저장된 DB번호 Temp영역에 저장
      L     #Order_Data_Send_DB_No;
      T     #ORDER_DATA_SEND_DB;

      OPN   DI [#FAC_LOG_DB]; //FAC Log 저장 DB를 Instance DB로 Open

NETWORK
TITLE =현 공정 차종 데이터를 FAC Log저장용 DB로 Move

      CALL FC   504 (
           SourceData_DB            := #LINE_PRESENT_DATA_DB,
           SourceStart_Add          := #Line_Present_Data_Byte,
           BLKMOV_Byte_Length       := 16,
           DestData_DB              := #FAC_LOG_DB,
           DestStart_Add            := 16);
      NOP   0;
NETWORK
TITLE =현재 공정의 VIN No(4자리) 취출(미완성 부분)
//DIW17,18=FAC Log 저장 DB의 현재 공정 VIN No. 저장 영역
//#Present_STA_VIN4=취출한 데이터를 임시 저장
      A(    ;
      L     DIW   17;
      L     DIW   18;
      OW    ;
      T     #Present_STA_VIN4;
      SET   ;
      SAVE  ;
      CLR   ;
      A     BR;
      )     ;
      JNB   M001;
      L     DIW   18;
      T     #Present_STA_VIN4;
M001: NOP   0;
NETWORK
TITLE =설정된 Terminal번호를 이용하여 FAC DB에서 시작 Byte 계산

      A(    ;
      L     60;
      L     #Terminal;
      *I    ;
      T     #FAC_DB_Start_Byte_temp;
      AN    OV;
      SAVE  ;
      CLR   ;
      A     BR;
      )     ;
      JNB   M002;
      L     #FAC_DB_Start_Byte_temp;
      L     60;
      -I    ;
      T     #FAC_DB_Start_Byte;
M002: NOP   0;
NETWORK
TITLE =Terminal번호(1~16)가 잘못 설정될 경우 OB로 Return

      O(    ;
      L     0;
      L     #Terminal;
      ==I   ;
      )     ;
      O(    ;
      L     16;
      L     #Terminal;
      <I    ;
      )     ;
      SAVE  ;
      BEC   ;
NETWORK
TITLE =해당 Terminal의 DB번호를 이용하여 DB Open 및 Accu1에 Byte저장

      OPN   DB [#FAC_DB];
      L     #FAC_DB_Start_Byte;
      SLW   3;
      LAR1  ;
NETWORK
TITLE =항상ON

      O     #NORMAL_ON;
      ON    #NORMAL_ON;
      =     #NORMAL_ON;
NETWORK
TITLE =FAC-PLC 통신 CHECK1
//DBW00=(FAC=11,PLC=1로 set)
//DIW32=(2초 시간 계산을 위한 Memory)
//DIW34=(10초 시간 계산을 위한 Memory)
      L     #FAC_DB_Start_Byte;
      SLW   3;
      LAR1  ;
      A(    ;
      A(    ; //DBW    0
      A(    ;
      A     #Flicker_1s;
      A(    ;
      L     11;
      L     DBW [AR1,P#0.0];
      ==I   ;
      )     ;
      FP    DIX   58.0;
      JNB   M003;
      L     1;
      L     DIW   32;
      +I    ;
      T     DIW   32;
      AN    OV;
      SAVE  ;
      CLR   ;
M003: A     BR;
      )     ;
      A(    ;
      L     2;
      L     DIW   32;
      <I    ;
      )     ; //DBW    0
      JNB   M005;
      L     #FAC_DB_Start_Byte;
      SLW   3;
      LAR1  ;
      L     1;
      T     DBW [AR1,P#0.0];
      SET   ;
      SAVE  ;
      CLR   ;
M005: A     BR;
      )     ;
      JNB   M006;
      L     0;
      T     DIW   32;
      SET   ;
      SAVE  ;
      CLR   ;
M006: A     BR;
      )     ;
      JNB   M007;
      L     0;
      T     DIW   34;
M007: NOP   0;
NETWORK
TITLE =FAC-PLC 통신 CHECK2
//DBW00=(FAC=11,PLC=1로 set)
//DIW32=(2초 시간 계산을 위한 Memory)
//DIW34=(10초 시간 계산을 위한 Memory)
      L     #FAC_DB_Start_Byte;
      SLW   3;
      LAR1  ;
      A     #Flicker_1s; //DBW    0
      A(    ;
      L     11;
      L     DBW [AR1,P#0.0];
      <>I   ;
      )     ;
      A(    ;
      L     10;
      L     DIW   34;
      >I    ;
      )     ;
      FP    DIX   58.1;
      JNB   M004;
      L     1;
      L     DIW   34;
      +I    ;
      T     DIW   34;
M004: NOP   0;
NETWORK
TITLE =FAC-PLC 통신 CHECK3
//DBW0의 데이터가 10초 동안 '11'로 바뀌지 않으면 통신이상
      L     10;
      L     DIW   34;
      <=I   ;
      =     #Communication_Error;
NETWORK
TITLE =생산지시 ON MODE
//DBW2=생산지시 on/off 선택 정보 저장 영역(1=ON,0=OFF)


      L     #FAC_DB_Start_Byte;
      SLW   3;
      LAR1  ;
      A     #ONLINE_Mode_Select; //DBW    2
      JNB   M008;
      L     1;
      T     DBW [AR1,P#2.0];
M008: NOP   0;
NETWORK
TITLE =생산지시 OFF MODE
//DBW2=생산지시 on/off 선택 정보 저장 영역(1=ON,0=OFF)
      L     #FAC_DB_Start_Byte;
      SLW   3;
      LAR1  ;
      AN    #ONLINE_Mode_Select; //DBW    2
      JNB   M009;
      L     0;
      T     DBW [AR1,P#2.0];
M009: NOP   0;
NETWORK
TITLE =공정 작업완료 SET 정보 전송
//DBW4=해당 공정 작업 완료 정보 저장 영역(1=ON,0=OFF)
      L     #FAC_DB_Start_Byte;
      SLW   3;
      LAR1  ;

      A     #Work_Complete;
      FP    DIX   58.2;
      JNB   M010;
      L     1;
      T     DBW [AR1,P#4.0]; //DBW    4
M010: NOP   0;
NETWORK
TITLE =공정 작업완료 RESET시 차종 요청 카운터 횟수 Clear
//DBW6=차종 설정 요구 발생 횟수 저장 영역
      L     #FAC_DB_Start_Byte;
      SLW   3;
      LAR1  ;

      A(    ;
      A     #Work_Complete;

      FN    DIX   58.3;
      JNB   M011;
      L     0;
      T     DBW [AR1,P#4.0]; //DBW    4
      SET   ;
      SAVE  ;
      CLR   ;
M011: A     BR;
      )     ;
      JNB   M012;
      L     #FAC_DB_Start_Byte;
      SLW   3; //DBW    6
      LAR1  ;
      L     0;
      T     DBW [AR1,P#6.0];
M012: NOP   0;
NETWORK
TITLE =공정 작업완료 SET시 log저장 함수 호출
//FC2=LOG 저장용 함수
      L     #FAC_DB_Start_Byte;
      SLW   3;
      LAR1  ;

      A(    ;
      L     1;
      L     DBW [AR1,P#4.0]; //DBW    4
      ==I   ;
      )     ;
      FP    DIX   58.4;
      JNB   M013;
      CALL FC   502 (
           FAC_Log_DB_NO            := #FAC_LOG_DB,
           LOG_INDEX                := W#16#400,
           LOG_DEC_DATA             := 0,
           LOG_BCD_DATA             := #Present_STA_VIN4);
M013: NOP   0;
NETWORK
TITLE =공정 작업완료 RESET시 log저장 함수 호출
//FC2=LOG 저장용 함수
      L     #FAC_DB_Start_Byte;
      SLW   3;
      LAR1  ;

      A(    ;
      L     0;
      L     DBW [AR1,P#4.0]; //DBW    4
      ==I   ;
      )     ;
      FP    DIX   58.5;
      JNB   M014;
      CALL FC   502 (
           FAC_Log_DB_NO            := #FAC_LOG_DB,
           LOG_INDEX                := W#16#500,
           LOG_DEC_DATA             := 0,
           LOG_BCD_DATA             := #Present_STA_VIN4);
M014: NOP   0;
NETWORK
TITLE =차종 설정 요청 정보 전송
//DBW22=차종 설정 요청 정보 '1'로 set
//DBW6=차종 설정 요구 발생 횟수 저장 영역
//
//#Data_Shift_Condition=해당 공정의 차종이 다음 공정으로 전송되는 조건
//
//1.생산지시용 데이터 수신 영역을 모두 삭제
//2.차종 설정 요청 발생 횟수 카운터 1증가
//3.차종 설정 요청 정보 '1'로 set

      L     #FAC_DB_Start_Byte;
      SLW   3;
      LAR1  ;

      A(    ;
      A(    ;
      A(    ;
      A(    ; //DIX   58.6
      A(    ;
      A     #Data_Shift_Condition;
      AN    DIX   61.0; //DBW   22
      FP    DIX   58.6;
      JNB   M015;
      L     40;
      L     #FAC_DB_Start_Byte;
      +I    ;
      T     #BLKMove_Sourcstart_point;
      AN    OV;
      SAVE  ; //DBW    6
      CLR   ;
M015: A     BR; //DBW    6
      )     ;
      JNB   M016;
      L     #FAC_DB_Start_Byte;
      SLW   3;
      LAR1  ;
      CALL FC   504 (
           SourceData_DB            := #FAC_DB,
           SourceStart_Add          := #BLKMove_Sourcstart_point,
           BLKMOV_Byte_Length       := 16,
           DestData_DB              := #FAC_LOG_DB,
           DestStart_Add            := 0);
M016: A     BR;
      )     ;
      JNB   M017;
      L     24;
      L     #FAC_DB_Start_Byte;
      +I    ;
      T     #Fill_start_point;
      AN    OV;
      SAVE  ;
      CLR   ;
M017: A     BR;
      )     ;
      JNB   M021;
      L     #FAC_DB_Start_Byte;
      SLW   3;
      LAR1  ;
      CALL FC   503 (
           Data_DB                  := #FAC_DB,
           Data_Length              := 32,
           FillStart_Add            := #Fill_start_point,
           Fill_Data                := B#16#0);
M021: A     BR;
      )     ;
      JNB   M022;
      L     #FAC_DB_Start_Byte;
      SLW   3;
      LAR1  ;
      L     1;
      L     DBW [AR1,P#6.0];
      +I    ;
      T     DBW [AR1,P#6.0];
      AN    OV;
      SAVE  ;
      CLR   ;
M022: A     BR;
      )     ;
      JNB   M023;
      L     #FAC_DB_Start_Byte;
      SLW   3;
      LAR1  ;
      L     1;
      T     DBW [AR1,P#22.0];
M023: A     BR;
      R     DIX   52.2;
      R     DIX   52.3;
NETWORK
TITLE =차종 설정 요청 정보 전송
//DBW22=차종 설정 요청 정보 '1'로 set
//DBW6=차종 설정 요구 발생 횟수 저장 영역
//
//#Data_Shift_Condition=해당 공정의 차종이 다음 공정으로 전송되는 조건
//
//1.생산지시용 데이터 수신 영역을 모두 삭제
//2.차종 설정 요청 발생 횟수 카운터 1증가
//3.차종 설정 요청 정보 '1'로 set

      L     #FAC_DB_Start_Byte;
      SLW   3;
      LAR1  ;

      A(    ;
      L     DBW [AR1,P#6.0];
      T     #Data_SET_Req_Count; //DBW   22
      SET   ;
      SAVE  ;
      CLR   ;
      A     BR;
      )     ;
      JNB   M024;
      L     #FAC_DB_Start_Byte;
      SLW   3;
      LAR1  ;
      L     DBW [AR1,P#8.0];
      T     #Final_Send_VIN;
M024: NOP   0;
NETWORK
TITLE =차종 설정 요청 발생 횟수 정보를 Temp영역으로 전송
//DBW6=차종 설정 요구 발생 횟수 저장 영역
//#Data_SET_Req_Count==차종 설정 요구 발생 횟수 임시(Log저장용) 저장 영역
      L     #FAC_DB_Start_Byte;
      SLW   3;
      LAR1  ;

      A(    ;
      L     1; //DBW    6
      L     DBW [AR1,P#22.0];
      ==I   ;
      )     ;
      FP    DIX   58.7;
      JNB   M025;
      CALL FC   502 (
           FAC_Log_DB_NO            := #FAC_LOG_DB,
           LOG_INDEX                := W#16#200,//DBW    8
           LOG_DEC_DATA             := #Data_SET_Req_Count,
           LOG_BCD_DATA             := #Final_Send_VIN);
M025: NOP   0;
NETWORK
TITLE =차종 설정 요청 정보 Log 저장 함수 호출
//DBW22=차종 설정 요청 정보 '1'로 set
      L     #FAC_DB_Start_Byte;
      SLW   3;
      LAR1  ;

      L     DBW [AR1,P#22.0];
      T     #FAC_Data_NewValue;
      NOP   0; //DBW   22
NETWORK
TITLE =차종 설정 요청 정보의 데이터 변경 확인1
//DIW36=이전에 저장된 차종 설정 요청 정보의 데이터 저장 영역
//DBW22=현재 차종 설정 요청 정보의 데이터 저장 영역
//#FAC_Data_OldValue=이전에 저장된 차종 설정 요청 정보의 데이터 임시 저장 영역
//#FAC_Data_NewValue=현재 차종 설정 요청 정보의 데이터 저장 영역
      L     #FAC_DB_Start_Byte; //DBW   22
      SLW   3;
      LAR1  ;
      L     DBW [AR1,P#24.0];
      T     #Present_RCV_VIN4;
      NOP   0;
NETWORK
TITLE =현재 수신된 VIN No. 4자리 취출용(미완성 부분)
//DBW24~26=현재 수신된 정보의 Vin No.저장 영역
//#Present_RCV_VIN4=현재 수신된 정보의 Vin No.임시(Log저장용) 저장 영역
      L     #FAC_DB_Start_Byte; //DBW   24
      SLW   3;
      LAR1  ;
      A(    ;
      L     0;
      L     DBW [AR1,P#22.0];
      <>I   ;
      )     ;
      A(    ;
      L     1;
      L     DBW [AR1,P#22.0];
      <>I   ;
      )     ;
      A(    ;
      L     DIW   36;
      L     DBW [AR1,P#22.0];
      <>I   ;
      )     ;
      FP    DIX   59.0;
      =     L     32.0;
      A     L     32.0;
      A(    ;
      L     99;
      L     DBW [AR1,P#22.0];
      <>I   ;
      )     ;
      A(    ;
      L     100;
      L     DBW [AR1,P#22.0];
      <>I   ;
      )     ;
      JNB   M026;
      CALL FC   502 (
           FAC_Log_DB_NO            := #FAC_LOG_DB,
           LOG_INDEX                := W#16#300,
           LOG_DEC_DATA             := #FAC_Data_NewValue,
           LOG_BCD_DATA             := #Present_RCV_VIN4);
M026: NOP   0;
      A     L     32.0;
      A(    ;
      L     100;
      L     DBW [AR1,P#22.0];
      ==I   ;
      )     ;
      JNB   M027;
      CALL FC   502 (
           FAC_Log_DB_NO            := #FAC_LOG_DB,
           LOG_INDEX                := W#16#600,
           LOG_DEC_DATA             := #FAC_Data_NewValue,
           LOG_BCD_DATA             := #Present_RCV_VIN4);
M027: NOP   0;
NETWORK
TITLE =차종 설정 요청 정보 내용 변경 확인 및 LOG 저장
//#FAC_Data_OldValue=이전에 저장된 차종 설정 요청 정보의 데이터 임시 저장 영역
//#FAC_Data_NewValue=현재 차종 설정 요청 정보의 데이터 저장 영역
//#FAC_Data_OldValue 와 #FAC_Data_NewValue를 비교하여 다르면 #FAC_Data_NewValue를
//#FAC_Data_OldValue에 전송하고 Log함수를 호출하여 정보를 저장한다.
//
//-#FAC_Data_NewValue(DBW22) 데이터 속성
//'1'=차종 설정 요청(PLC set)
//'11'=차종 설정 요청 처리 정상(FAC set)
//'12'~'98'=차종 설정 요청 처리 이상(FAC set)
//'99'=서열 데이터 부족(FAC set)
//'100'=차종 강제(수동) 설정(FAC set)
//dix54.7 pls삭제함
      L     #FAC_DB_Start_Byte;
      SLW   3;
      LAR1  ;

      A(    ;
      A(    ;
      L     100; //DBW   22
      L     DBW [AR1,P#22.0];
      ==I   ;
      )     ;
      FP    DIX   59.1;
      JNB   M028; //DBW   22
      L     0;
      T     DBW [AR1,P#6.0];
      SET   ;
      SAVE  ;
      CLR   ; //DBW   22
M028: A     BR;
      )     ;
      JNB   M029;
      CALL FC   503 (
           Data_DB                  := #FAC_LOG_DB,
           Data_Length              := 16,
           FillStart_Add            := 0,
           Fill_Data                := B#16#0);//DBW   22
M029: A     BR;
      S     DIX   61.0;
NETWORK
TITLE =차종 강제 설정시 차종 설정 요청 카운터 및 수신 비교 정보 clear
//DBW22=차종 설정 요청 정보 ('100'=강제(수동)설정)
//DBW6=차종 설정 요구 발생 횟수 저장 영역
      A     #Work_Complete;
      FN    DIX   61.1;
      R     DIX   61.0;

NETWORK
TITLE =

      L     #FAC_DB_Start_Byte;
      SLW   3;
      LAR1  ;

      A(    ;
      O(    ;
      L     11;
      L     DBW [AR1,P#22.0];
      ==I   ;
      )     ;
      O(    ;
      L     99;
      L     DBW [AR1,P#22.0];
      ==I   ;
      )     ;
      )     ;
      FP    DIX   59.2;
      A(    ;
      L     L#0;
      L     DID    0;
      <>D   ;
      )     ;
      =     L     32.0;
      A     L     32.0;
      A(    ;
      L     DBD [AR1,P#24.0];
      L     DBD [AR1,P#8.0];
      <>D   ;
      )     ;
      S     DIX   52.0;
      A     L     32.0;
      A(    ;
      L     DBD [AR1,P#24.0];
      L     DID    0;
      ==D   ;
      )     ;
      A(    ;
      L     DBD [AR1,P#28.0];
      L     DID    4;
      ==D   ;
      )     ;
      A(    ;
      L     DBD [AR1,P#32.0];
      L     DID    8;
      ==D   ;
      )     ;
      A(    ;
      L     DBD [AR1,P#36.0];
      L     DID   12;
      ==D   ;
      )     ;
      S     DIX   52.1;
      A     L     32.0;
      BLD   102;
      S     DIX   61.2;
NETWORK
TITLE =현재 수신 데이터를 VIN No를 이용하여 이상 여부 확인
//DBW22=차종 설정 요청 정보 ('11'=FAC 정상 처리)
//DBD24~28=서열 데이터 VIN No. 수신 영역(현재 생산)
//DIW0~4=수신 데이터 비교를 위해 이전에 수신된 데이터에서 다음 수신 예정 정보를
//저장해 놓은
//       영역
//DIX52.0=중복 데이터가 아님
//DIX52.1=이전에 수신된 정보와 비교하여 VIN No.가 일치함
      L     #FAC_DB_Start_Byte;
      SLW   3;
      LAR1  ;
      A(    ;
      O(    ;
      L     11;
      L     DBW [AR1,P#22.0]; //DBW   22
      ==I   ;
      )     ;
      O(    ;
      L     99;
      L     DBW [AR1,P#22.0]; //DBW   22
      ==I   ;
      )     ;
      )     ;
      A     DIX   52.0;
      A     DIX   52.1;
      O(    ;
      L     100;
      L     DBW [AR1,P#22.0];
      ==I   ;
      )     ;
      O(    ;
      L     0;
      L     #ORDER_DATA_SEND_DB; //DBD   24
      ==I   ; //DBD    8
      )     ;
      O     ;
      A(    ;
      L     L#0;
      L     DID    0;
      ==D   ; //DBD   24
      )     ;
      A(    ;
      L     L#0;
      L     DID    4;
      ==D   ;
      )     ;
      S     DIX   52.2;


NETWORK
TITLE =수신 데이터 비교 결과= 정상(0813수정)
//DBW22=차종 설정 요청 정보 ('11'=FAC 설정 요청 정상처리,'100'=강제(수동)설정)
//DIX52.0=중복 데이터가 아님
//DIX52.1=이전에 수신된 정보와 비교하여 VIN No.가 일치함
//DIX52.2=수신 데이터 비교 결과 정상
      L     #FAC_DB_Start_Byte;
      SLW   3;
      LAR1  ;

      A(    ;
      O(    ;
      L     11;
      L     DBW [AR1,P#22.0]; //DBW   22
      ==I   ;
      )     ;
      O(    ;
      L     99;
      L     DBW [AR1,P#22.0]; //DBW   22
      ==I   ;
      )     ;
      )     ;
      A(    ;
      ON    DIX   52.0;
      ON    DIX   52.1;
      )     ;
      A(    ; //DBW   22
      L     L#0;
      L     DBD [AR1,P#24.0];
      <>D   ;
      )     ;
      A     DIX   61.2;
      A(    ;
      L     0;
      L     #Order_Data_Send_DB_No;
      <>I   ;
      )     ;
      A(    ;
      L     L#0;
      L     DID    0;
      <>D   ;
      )     ;
      A(    ;
      L     L#0;
      L     DID    4;
      <>D   ;

      )     ;
      S     DIX   52.3;
NETWORK
TITLE =수신 데이터 비교 결과= 이상(0813수정)
//DBW22=차종 설정 요청 정보 ('11'=FAC 설정 요청 정상처리,'100'=강제(수동)설정)
//DIX52.0=중복 데이터가 아님
//DIX52.1=이전에 수신된 정보와 비교하여 VIN No.가 일치함
//DIX52.2=수신 데이터 비교 결과 정상
      L     #FAC_DB_Start_Byte;
      SLW   3;
      LAR1  ;

      A(    ;
      L     99;
      L     DBW [AR1,P#22.0];
      ==I   ; //DBW   22
      )     ;
      FP    DIX   59.3;
      S     DIX   52.6;
NETWORK
TITLE =서열 데이터 부족 출력 Set
//응답코드가 '99'일때 설비쪽으로 알려주기 위한 Logic
//응답코드 '99'=서열 데이터 부족
//DIX52.3=서열 데이터 부족 Alarm 출력 보조
      L     #FAC_DB_Start_Byte;
      SLW   3;
      LAR1  ;

      A     DIX   52.6;
      A(    ;
      O(    ; //DBW   22
      L     11;
      L     DBW [AR1,P#22.0];
      ==I   ;
      )     ;
      O(    ;
      L     100;
      L     DBW [AR1,P#22.0];
      ==I   ;
      )     ;
      )     ;
      R     DIX   52.6;
NETWORK
TITLE =서열 데이터 부족 출력 Reset
//응답코드가 '99'에서 정상적인 응답코드 수신('11') 또는 강제설정시('100') Reset
//응답코드  '11'=차종설정요청('1')에 대한 정상 처리 코드
//응답코드 '100'=차종 강제 설정 처리 코드
//DIX52.3=서열 데이터 부족 Alarm 출력 보조
      L     #FAC_DB_Start_Byte;
      SLW   3;
      LAR1  ;

      AN    DIX   52.2;
      A     DIX   52.3;
      A(    ;
      L     0;
      L     #ORDER_DATA_SEND_DB; //DBW   22
      <>I   ;
      )     ;
      FP    DIX   59.5;
      =     L     32.0;
      A     L     32.0; //DBW   22
      AN    DIX   52.0;
      JNB   M030;
      L     1;
      T     DBW [AR1,P#12.0];
M030: NOP   0;
      A     L     32.0;
      A     DIX   52.0;
      AN    DIX   52.1;
      JNB   M031;
      L     2;
      T     DBW [AR1,P#12.0];
M031: NOP   0;
NETWORK
TITLE =수신 데이터 비교 결과 이상시 FAC로 통보(0813수정)
//DBW22=차종 설정 요청 정보 ('11'=FAC 설정 요청 정상 처리,'100'=강제(수동)설정)
//DBW12=수신 차종 비교 이상 정보 저장 영역(1=중복,2=이전 데이터와 비교 결과
//불일치)
//DIX52.0=중복 데이터가 아님
//DIX52.1=이전에 수신된 정보와 비교하여 VIN No.가 일치함
//DIX52.2=수신 데이터 비교 결과 정상
//#Data_Request=설비측에 차종 데이터를 요청하는 신호
      L     #FAC_DB_Start_Byte;
      SLW   3;
      LAR1  ;

      A(    ;
      A(    ;
      O     DIX   52.2;
      O     DIX   52.3;
      )     ;
      A(    ;
      L     1;
      L     DBW [AR1,P#22.0];
      <>I   ;
      )     ;
      A(    ;
      L     3;
      L     DBW [AR1,P#22.0];
      <>I   ; //DBW   12
      )     ;
      FP    DIX   59.4;
      JNB   M032;
      L     3;
      T     DBW [AR1,P#22.0];
      SET   ;
      SAVE  ; //DBW   12
      CLR   ;
M032: A     BR;
      )     ;
      JNB   M033;
      L     #FAC_DB_Start_Byte;
      SLW   3;
      LAR1  ;
      L     DBW [AR1,P#22.0];
      T     DIW   36;
      SET   ;
      SAVE  ;
      CLR   ;
M033: A     BR;
      R     DIX   52.0;
      R     DIX   52.1;
      R     DIX   61.2;
NETWORK
TITLE =응답코드에 대한 처리 완료 후 응답 코드를 '3'으로 변환

      AN    DIX   52.2;
      A     DIX   52.3;
      O     DIX   52.6;

      =     #Data_Error;
NETWORK
TITLE =수신 데이터 비교 결과 이상시 설비측으로 통보
//#Data_Request=설비측에 차종 데이터를 요청하는 신호
//DIX52.2=수신 데이터 비교 결과 정상
//DBW22=차종 설정 요청 정보 ('1'=설정 요청,'11'=FAC 설정 요청 정상처리,
//                         '100'=강제(수동)설정)
//#Data_Error=함수 외부로 출력되는 Bit 신호
      L     #FAC_DB_Start_Byte;
      SLW   3;
      LAR1  ;
      A(    ;
      L     3;
      L     DBW [AR1,P#22.0];
      ==I   ;
      )     ;
      A     DIX   52.2;
      =     L     32.0;
      A     L     32.0;
      BLD   102;
      =     DIX   52.7;
      A     L     32.0;
      JNB   M034;
      L     0;
      T     DBW [AR1,P#12.0];
M034: NOP   0;
NETWORK
TITLE =수신 데이터 비교 정상
//DBW22=차종 설정 요청 정보 ('11'=FAC 설정 요청 정상 처리,'100'=강제(수동)설정)
//DIX52.2=수신 데이터 비교 결과 정상
//DIX52.4=수신 데이터 비교 결과 정상이므로 설비측으로 데이터 전송 가능
//DBW12=수신 차종 비교 이상 정보 저장 영역(1=중복,2=이전 데이터와 비교 결과
//불일치)
      L     #FAC_DB_Start_Byte;
      SLW   3;
      LAR1  ;

      A(    ;
      L     DBW [AR1,P#24.0];
      T     DIW 1102; //DBW   22
      SET   ;
      SAVE  ;
      CLR   ;
      A     BR;
      )     ;
      JNB   M035;
      L     #FAC_DB_Start_Byte;
      SLW   3;
      LAR1  ;
      L     DBW [AR1,P#26.0];
      T     DIW 1100; //DBW   12
M035: NOP   0;
NETWORK
TITLE =

      L     #FAC_DB_Start_Byte;
      SLW   3;
      LAR1  ;

      A(    ;
      A(    ; //DBW   24
      A(    ;
      L     DBB [AR1,P#28.0];
      T     DIB 1105;
      SET   ;
      SAVE  ;
      CLR   ;
      A     BR;
      )     ; //DBW   26
      JNB   M036;
      L     #FAC_DB_Start_Byte;
      SLW   3;
      LAR1  ;
      L     DBB [AR1,P#29.0];
      T     DIB 1104;
      SET   ;
      SAVE  ;
      CLR   ;
M036: A     BR;
      )     ;
      JNB   M018;
      L     #FAC_DB_Start_Byte;
      SLW   3;
      LAR1  ;
      L     DBB [AR1,P#30.0];
      T     DIB 1107;
      SET   ;
      SAVE  ;
      CLR   ;
M018: A     BR;
      )     ;
      JNB   M019;
      L     #FAC_DB_Start_Byte;
      SLW   3;
      LAR1  ;
      L     DBB [AR1,P#31.0];
      T     DIB 1106;
M019: NOP   0;
NETWORK
TITLE =

      L     #FAC_DB_Start_Byte;
      SLW   3;
      LAR1  ;

      A(    ;
      A(    ;
      A(    ;
      L     DBB [AR1,P#32.0]; //DBB   28
      T     DIB 1109;
      SET   ;
      SAVE  ;
      CLR   ;
      A     BR;
      )     ;
      JNB   M020;
      L     #FAC_DB_Start_Byte; //DBB   29
      SLW   3;
      LAR1  ;
      L     DBB [AR1,P#33.0];
      T     DIB 1108;
      SET   ;
      SAVE  ;
      CLR   ;
M020: A     BR; //DBB   30
      )     ;
      JNB   M037;
      L     #FAC_DB_Start_Byte;
      SLW   3;
      LAR1  ;
      L     DBB [AR1,P#34.0];
      T     DIB 1111;
      SET   ; //DBB   31
      SAVE  ;
      CLR   ;
M037: A     BR;
      )     ;
      JNB   M038;
      L     #FAC_DB_Start_Byte;
      SLW   3;
      LAR1  ;
      L     DBB [AR1,P#35.0];
      T     DIB 1110;
M038: NOP   0;
NETWORK
TITLE =

      L     #FAC_DB_Start_Byte;
      SLW   3;
      LAR1  ;

      A(    ;
      A(    ;
      A(    ;
      L     DBB [AR1,P#36.0]; //DBB   32
      T     DIB 1113;
      SET   ;
      SAVE  ;
      CLR   ;
      A     BR;
      )     ;
      JNB   M039;
      L     #FAC_DB_Start_Byte; //DBB   33
      SLW   3;
      LAR1  ;
      L     DBB [AR1,P#37.0];
      T     DIB 1112;
      SET   ;
      SAVE  ;
      CLR   ;
M039: A     BR; //DBB   34
      )     ;
      JNB   M040;
      L     #FAC_DB_Start_Byte;
      SLW   3;
      LAR1  ;
      L     DBB [AR1,P#38.0];
      T     DIB 1115;
      SET   ; //DBB   35
      SAVE  ;
      CLR   ;
M040: A     BR;
      )     ;
      JNB   M041;
      L     #FAC_DB_Start_Byte;
      SLW   3;
      LAR1  ;
      L     DBB [AR1,P#39.0];
      T     DIB 1114;
M041: NOP   0;
NETWORK
TITLE =

      L     #FAC_DB_Start_Byte;
      SLW   3;
      LAR1  ;

      A(    ;
      A     #Flicker_1s;
      A     #Data_Request;
      FP    DIX   61.3; //DBB   36
      JNB   M058;
      L     1;
      L     DIW   38;
      +I    ;
      T     DIW   38;
      AN    OV;
      SAVE  ;
      CLR   ; //DBB   37
M058: A     BR;
      )     ;
      A(    ;
      L     2;
      L     DIW   38;
      <I    ;
      )     ;
      S     DIX   61.4; //DBB   38
NETWORK
TITLE =

      L     #FAC_DB_Start_Byte;
      SLW   3;
      LAR1  ;

      AN    #Data_Request;
      JNB   M059;
      L     0;
      T     DIW   38;
      SET   ;
      SAVE  ;
      CLR   ;
M059: A     BR;
      R     DIX   61.4;
NETWORK
TITLE =

      L     #FAC_DB_Start_Byte;
      SLW   3;
      LAR1  ;

      A(    ;
      L     1;
      L     DBW [AR1,P#2.0];
      ==I   ;
      )     ;
      A(    ;
      L     3;
      L     DBW [AR1,P#22.0];
      ==I   ;


      )     ;
      A     #Data_Request;
      A     DIX   52.7;
      A     DIX   61.4;
      =     L     32.0;
      A     L     32.0;
      JNB   M042;
      CALL FC   504 (
           SourceData_DB            := #FAC_LOG_DB,
           SourceStart_Add          := 1100,
           BLKMOV_Byte_Length       := 16,
           DestData_DB              := #Order_Data_Send_DB_No,
           DestStart_Add            := #Order_Data_Send_DB_Byte);
M042: NOP   0;
      A(    ;
      A(    ;
      A     L     32.0;
      JNB   M043;
      L     24;
      L     #FAC_DB_Start_Byte;
      +I    ;
      T     #BLKMove_Sourcstart_point;
      AN    OV;
      SAVE  ;
      CLR   ;
M043: A     BR;
      )     ;
      JNB   M044;
      L     8;
      L     #FAC_DB_Start_Byte;
      +I    ;
      T     #BLKMove_Deststart_point;
      AN    OV;
      SAVE  ;
      CLR   ;
M044: A     BR;
      )     ;
      JNB   M045;
      CALL FC   504 (
           SourceData_DB            := #FAC_DB,
           SourceStart_Add          := #BLKMove_Sourcstart_point,
           BLKMOV_Byte_Length       := 4,
           DestData_DB              := #FAC_DB,
           DestStart_Add            := #BLKMove_Deststart_point);
M045: NOP   0;
      A(    ;
      A     L     32.0;
      JNB   M046;
      L     40;
      L     #FAC_DB_Start_Byte;
      +I    ;
      T     #BLKMove_Sourcstart_point;
      AN    OV;
      SAVE  ;
      CLR   ;
M046: A     BR;
      )     ;
      JNB   M047;
      CALL FC   504 (
           SourceData_DB            := #FAC_DB,
           SourceStart_Add          := #BLKMove_Sourcstart_point,
           BLKMOV_Byte_Length       := 16,
           DestData_DB              := #FAC_LOG_DB,
           DestStart_Add            := 0);
M047: NOP   0;
NETWORK
TITLE =설비측 차종 요청 ON시 데이터 전송
//DBW22=생산지시 ON/OFF 선택 정보(1=ON)
//#Data_Request=함수로 입력된 신호(설비측에서 차종 데이터 요구)
//DIX50.3=수신 데이터 비교 결과 정상이므로 설비측으로 데이터 전송 가능
//
//1.수신 데이터를 설비측으로 #Order_Data_Send_DB_No의
//#Order_Data_Send_DB_Byte부터
//  16Byte를 전송
//2.설비측으로 전송한 데이터에서 VIN No.(공정 최종 전송)를 DB에 저장
//3.다음에 수신할 데이터를 비교하기 위해 FAC Log저장용 DB에 전송
      L     #FAC_DB_Start_Byte;
      SLW   3;
      LAR1  ;

      A     #BType_Change_Set_Rst_PB;
      A(    ;
      L     1; //DBW    2
      L     DBW [AR1,P#22.0];
      <>I   ;
      )     ;
      A(    ;
      O     DIX   27.2; //DBW   22
      O     DIX   27.3;
      O     DIX   27.4;
      O     DIX   27.5;
      O     DIX   27.6;
      O     DIX   27.7;
      )     ;
      =     DIX   54.0;
      S     DIX   54.1;
NETWORK
TITLE = 현재 공정 차종 영역에서 운영 정보 bit확인
//DIX26.2~7=차종 영역 표준Map에서 운영정보용 BIT
//DIX54.0=차종 영역에 운영 정보 있음
//DIX54.1=차종 영역에 운영 정보 있음 기억
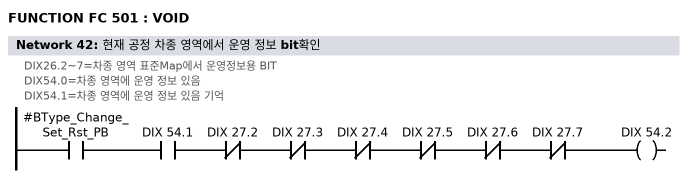
      A     #BType_Change_Set_Rst_PB;
      A     DIX   54.1;
      AN    DIX   27.2;

      AN    DIX   27.3;
//      A(
//      L     1
//    L     DBW [AR1,P#22.0]            //DBW   22
//  <>I
//      )
      AN    DIX   27.4;
      AN    DIX   27.5;
      AN    DIX   27.6;
      AN    DIX   27.7;
      =     DIX   54.2;
NETWORK
TITLE =수동으로 차종 삭제시 라인 정보 반영 확인
//#BType_Change_Set_Rst_PB=차종 수동으로 설정/리셋 버튼
//DIX54.1=차종 영역에 운영 정보 있음
//DIX54.3=차종 영역에 운영 정보 없음
//DIX26.2~7=차종 영역 표준Map에서 운영정보용 BIT
      L     #FAC_DB_Start_Byte;
      SLW   3;
      LAR1  ;
      A(    ;
      A(    ;
      A(    ;
      A(    ;
      A(    ;
      O     DIX   54.0;
      O     DIX   54.2;
      )     ;
      A(    ;
      L     1;
      L     DBW [AR1,P#22.0];
      <>I   ;
      )     ;
      FP    DIX   59.6;
      JNB   M060;
      L     1;
      T     DBW [AR1,P#20.0];
      SET   ;
      SAVE  ;
      CLR   ;
M060: A     BR;
      )     ;
      JNB   M061;
      CALL FC   503 (
           Data_DB                  := #FAC_LOG_DB,
           Data_Length              := 16,
           FillStart_Add            := 0,
           Fill_Data                := B#16#0);
M061: A     BR;
      )     ;
      JNB   M062;
      L     24;
      L     #FAC_DB_Start_Byte;
      +I    ;
      T     #Fill_start_point;
      AN    OV;
      SAVE  ;
      CLR   ;
M062: A     BR;
      )     ;
      JNB   M063;
      CALL FC   503 (
           Data_DB                  := #FAC_DB,
           Data_Length              := 32,
           FillStart_Add            := #Fill_start_point,
           Fill_Data                := B#16#0);
M063: A     BR;
      )     ;
      JNB   M064;
      L     #FAC_DB_Start_Byte;
      SLW   3;
      LAR1  ;
      L     0;
      T     DBW [AR1,P#12.0];
      SET   ;
      SAVE  ;
      CLR   ;
M064: NOP   0;
NETWORK
TITLE =운영 정보 있음 기억 clear
//DIX54.0=차종 영역에 운영 정보 있음 기억
//DIX54.2=차종 영역에 운영 정보 있음(바뀜) 검출
//DIX54.3=차종 영역에 운영 정보 없음
//#Data_Shift_Condition=해당 공정의 차종이 다음 공정으로 전송되는 조건
//DBW20=라인 현황 반영 요청 신호(PLC='1',FAC='11'로 SET)
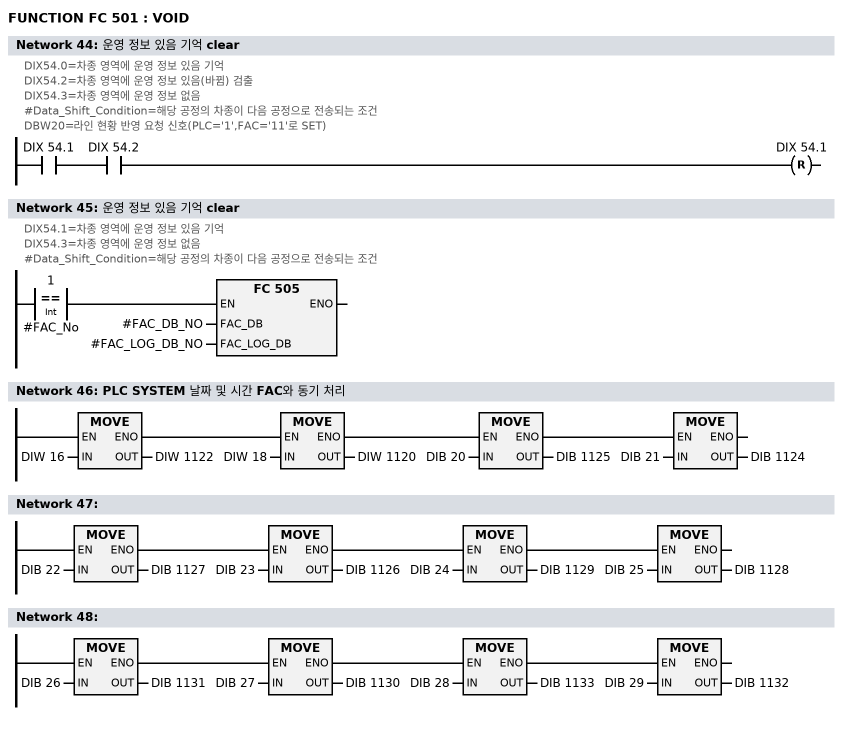
      A     DIX   54.1;
      A     DIX   54.2;
      R     DIX   54.1;

NETWORK
TITLE =운영 정보 있음 기억 clear
//DIX54.1=차종 영역에 운영 정보 있음 기억
//DIX54.3=차종 영역에 운영 정보 없음
//#Data_Shift_Condition=해당 공정의 차종이 다음 공정으로 전송되는 조건
      A(    ;
      L     1;
      L     #FAC_No;
      ==I   ;
      )     ;
      JNB   M048;
      CALL FC   505 (
           FAC_DB                   := #FAC_DB_NO,
           FAC_LOG_DB               := #FAC_LOG_DB_NO);

M048: NOP   0;
NETWORK
TITLE =PLC SYSTEM 날짜 및 시간 FAC와 동기 처리

      A(    ;
      A(    ;
      A(    ;
      L     DIW   16;
      T     DIW 1122;
      SET   ;
      SAVE  ;
      CLR   ;
      A     BR;
      )     ;
      JNB   M049;
      L     DIW   18;
      T     DIW 1120;
      SET   ;
      SAVE  ;
      CLR   ;
M049: A     BR;
      )     ;
      JNB   M050;
      L     DIB   20;
      T     DIB 1125;
      SET   ;
      SAVE  ;
      CLR   ;
M050: A     BR;
      )     ;
      JNB   M051;
      L     DIB   21;
      T     DIB 1124;
M051: NOP   0;
NETWORK
TITLE =

      A(    ;
      A(    ;
      A(    ;
      L     DIB   22;
      T     DIB 1127;
      SET   ;
      SAVE  ;
      CLR   ;
      A     BR;
      )     ;
      JNB   M052;
      L     DIB   23;
      T     DIB 1126;
      SET   ;
      SAVE  ;
      CLR   ;
M052: A     BR;
      )     ;
      JNB   M053;
      L     DIB   24;
      T     DIB 1129;
      SET   ;
      SAVE  ;
      CLR   ;
M053: A     BR;
      )     ;
      JNB   M054;
      L     DIB   25;
      T     DIB 1128;
M054: NOP   0;
NETWORK
TITLE =

      A(    ;
      A(    ;
      A(    ;
      L     DIB   26;
      T     DIB 1131;
      SET   ;
      SAVE  ;
      CLR   ;
      A     BR;
      )     ;
      JNB   M055;
      L     DIB   27;
      T     DIB 1130;
      SET   ;
      SAVE  ;
      CLR   ;
M055: A     BR;
      )     ;
      JNB   M056;
      L     DIB   28;
      T     DIB 1133;
      SET   ;
      SAVE  ;
      CLR   ;
M056: A     BR;
      )     ;
      JNB   M057;
      L     DIB   29;
      T     DIB 1132;
M057: NOP   0;
END_FUNCTION

FUNCTION FC 510 : VOID
TITLE =
VERSION : 0.1


VAR_INPUT
  FAC_No : INT ;	//Terminal No. 입력용
  FAC_DB_NO : INT ;	//생산지시용 DB 번호 입력용
  FAC_LOG_DB_NO : INT ;	//Terminal별 Log Data저장 DB 번호 입력용
  Line_Present_Data_DB_No : INT ;	//라인의 현재 공정 차종 영역이 저장된 DB번호 입력용
  Line_Present_Data_Byte : INT ;	//라인의 현재 공정 차종 영역이 저장된 DB의 Byte번호 입력용
  Order_Data_Send_DB_No : INT ;	//라인의 현재 공정에 서열 데이터를 수신할 DB번호 입력용
  Order_Data_Send_DB_Byte : INT ;	//라인의 현재 공정에 서열 데이터를 수신할 DB의 Byte번호 입력용
  ONLINE_Mode_Select : BOOL ;	//생산지시 ON/OFF 선택 스위치 또는 BIT 입력용
  Work_Complete : BOOL ;	//해당 공정의 작업완료 BIT 입력용
  Data_Shift_Condition : BOOL ;	//해당 공정에서 다음 공정으로 차종이 전송 되는 신호
  Data_Request : BOOL ;	//해당 공정에서 차종을 요구하는 신호
  BType_Change_Set_Rst_PB : BOOL ;	//수동으로 차종 Set/Reset 버튼
  Flicker_1s : BOOL ;	//PLC CPU에 정의된 1초 Clock용 신호
END_VAR
VAR_OUTPUT
  Communication_Error : BOOL ;	//terminal과 PLC간 통신 이상이 발생한 경우 출력
  Data_Error : BOOL ;	//Terminal에서 수신된 데이터에 이상이 발생한 경우 출력
END_VAR
VAR_TEMP
  Terminal : INT ;	//Terminal No. 저장 temp
  FAC_DB : INT ;	//생산지시용 DB 번호 저장 temp
  FAC_LOG_DB : INT ;	//Terminal별 Log Data저장 DB 번호 저장 temp
  LINE_PRESENT_DATA_DB : INT ;	//라인의 현재 공정 차종 영역이 저장된 DB번호 저장 temp
  ORDER_DATA_SEND_DB : INT ;	//라인의 현재 공정에 서열 데이터를 수신할 DB번호 저장 temp
  FAC_DB_Start_Byte_temp : INT ;	//Terminal별 FAC_DB의 시작 Byte 저장용
  FAC_DB_Start_Byte : INT ;	//Terminal별 FAC_DB의 시작 Byte 저장용
  NORMAL_ON : BOOL ;	//항상ON
  Present_RCV_VIN4 : WORD ;	//현재 수신된 데이터의 VIN No. 4자리
  Present_STA_VIN4 : WORD ;	//현재 공정 데이터의 VIN No. 4자리
  FAC_Data_NewValue : INT ;	//차종 설정 요청 정보의 데이터 변경 확인용 Temp1
  Final_Send_VIN : WORD ;	//차종 설정 요청 정보의 데이터 변경 확인용 Temp2
  Data_SET_Req_Count : INT ;	//차종 설정 요청 신호 발생 횟수 Temp
  Fill_start_point : INT ;
  BLKMove_Sourcstart_point : INT ;
  BLKMove_Deststart_point : INT ;
END_VAR
BEGIN
NETWORK
TITLE =FAC용 DB OPEN

      L     #FAC_No; //Terminal번호 Load
      T     #Terminal; //Terminal번호 Temp영역에 저장
      L     #FAC_DB_NO; //생산지시용 FAC DB번호 Load
      T     #FAC_DB; //생산지시용 FAC DB번호 Temp영역에 저장
      L     #FAC_LOG_DB_NO; //FAC Log 저장 DB번호 Load
      T     #FAC_LOG_DB; //FAC Log 저장 DB번호 Temp영역에 저장
      L     #Line_Present_Data_DB_No; //라인의 현재 공정 차종 영역이 저장된 DB번호 Load
      T     #LINE_PRESENT_DATA_DB; //라인의 현재 공정 차종 영역이 저장된 DB번호 Temp영역에 저장
      L     #Order_Data_Send_DB_No;
      T     #ORDER_DATA_SEND_DB;
      OPN   DI [#FAC_LOG_DB]; //FAC Log 저장 DB를 Instance DB로 Open

NETWORK
TITLE =현 공정 차종 데이터를 FAC Log저장용 DB로 Move

      CALL FC   504 (
           SourceData_DB            := #LINE_PRESENT_DATA_DB,
           SourceStart_Add          := #Line_Present_Data_Byte,
           BLKMOV_Byte_Length       := 16,
           DestData_DB              := #FAC_LOG_DB,
           DestStart_Add            := 16);
      NOP   0;
NETWORK
TITLE =현재 공정의 VIN No(4자리) 취출(미완성 부분)
//db241.dbw17,18=FAC Log 저장 DB의 현재 공정 VIN No. 저장 영역
//#Present_STA_VIN4=취출한 데이터를 임시 저장
      A(    ;
      L     DB241.DBW   17;
      L     DB241.DBW   18;
      OW    ;
      T     #Present_STA_VIN4;
      SET   ;
      SAVE  ;
      CLR   ;
      A     BR;
      )     ;
      JNB   _001;
      L     DB241.DBW   18;
      T     #Present_STA_VIN4;
_001: NOP   0;
NETWORK
TITLE =설정된 Terminal번호를 이용하여 FAC DB에서 시작 Byte 계산

      A(    ;
      L     60;
      L     #Terminal;
      *I    ;
      T     #FAC_DB_Start_Byte_temp;
      AN    OV;
      SAVE  ;
      CLR   ;
      A     BR;
      )     ;
      JNB   _002;
      L     #FAC_DB_Start_Byte_temp;
      L     60;
      -I    ;
      T     #FAC_DB_Start_Byte;
_002: NOP   0;
NETWORK
TITLE =Terminal번호(1~16)가 잘못 설정될 경우 OB로 Return

      O(    ;
      L     0;
      L     #Terminal;
      ==I   ;
      )     ;
      O(    ;
      L     16;
      L     #Terminal;
      <I    ;
      )     ;
      SAVE  ;
      BEC   ;
NETWORK
TITLE =해당 Terminal의 DB번호를 이용하여 DB Open 및 Accu1에 Byte저장

      OPN   DB [#FAC_DB];
      L     #FAC_DB_Start_Byte;
      SLW   3;
      LAR1  ;
NETWORK
TITLE =항상ON
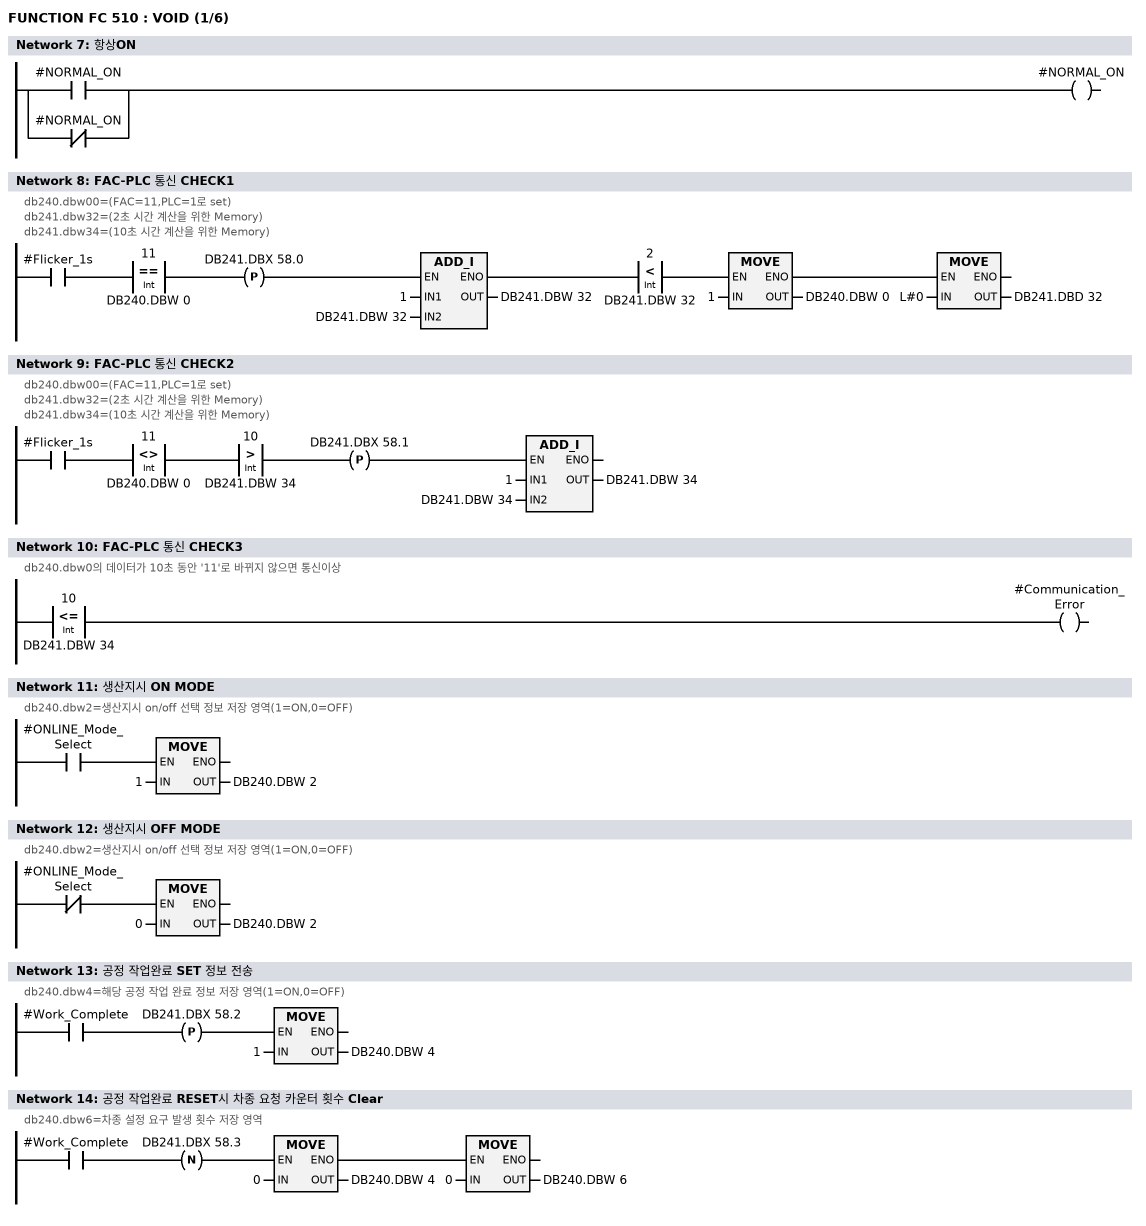

      O     #NORMAL_ON;
      ON    #NORMAL_ON;
      =     #NORMAL_ON;
NETWORK
TITLE =FAC-PLC 통신 CHECK1
//db240.dbw00=(FAC=11,PLC=1로 set)
//db241.dbw32=(2초 시간 계산을 위한 Memory)
//db241.dbw34=(10초 시간 계산을 위한 Memory)
      A(    ;
      A(    ;
      A     #Flicker_1s;
      A(    ;
      L     11;
      L     DB240.DBW    0;
      ==I   ;
      )     ;
      FP    DB241.DBX   58.0;
      JNB   _003;
      L     1;
      L     DB241.DBW   32;
      +I    ;
      T     DB241.DBW   32;
      AN    OV;
      SAVE  ;
      CLR   ;
_003: A     BR;
      )     ;
      A(    ;
      L     2;
      L     DB241.DBW   32;
      <I    ;
      )     ;
      JNB   _004;
      L     1;
      T     DB240.DBW    0;
      SET   ;
      SAVE  ;
      CLR   ;
_004: A     BR;
      )     ;
      JNB   _005;
      L     L#0;
      T     DB241.DBD   32;
_005: NOP   0;
NETWORK
TITLE =FAC-PLC 통신 CHECK2
//db240.dbw00=(FAC=11,PLC=1로 set)
//db241.dbw32=(2초 시간 계산을 위한 Memory)
//db241.dbw34=(10초 시간 계산을 위한 Memory)
      A     #Flicker_1s;
      A(    ;
      L     11;
      L     DB240.DBW    0;
      <>I   ;
      )     ;
      A(    ;
      L     10;
      L     DB241.DBW   34;
      >I    ;
      )     ;
      FP    DB241.DBX   58.1;
      JNB   _006;
      L     1;
      L     DB241.DBW   34;
      +I    ;
      T     DB241.DBW   34;
_006: NOP   0;
NETWORK
TITLE =FAC-PLC 통신 CHECK3
//db240.dbw0의 데이터가 10초 동안 '11'로 바뀌지 않으면 통신이상
      L     10;
      L     DB241.DBW   34;
      <=I   ;
      =     #Communication_Error;
NETWORK
TITLE =생산지시 ON MODE
//db240.dbw2=생산지시 on/off 선택 정보 저장 영역(1=ON,0=OFF)


      A     #ONLINE_Mode_Select;
      JNB   _007;
      L     1;
      T     DB240.DBW    2;
_007: NOP   0;
NETWORK
TITLE =생산지시 OFF MODE
//db240.dbw2=생산지시 on/off 선택 정보 저장 영역(1=ON,0=OFF)
      AN    #ONLINE_Mode_Select;
      JNB   _008;
      L     0;
      T     DB240.DBW    2;
_008: NOP   0;
NETWORK
TITLE =공정 작업완료 SET 정보 전송
//db240.dbw4=해당 공정 작업 완료 정보 저장 영역(1=ON,0=OFF)
      A     #Work_Complete;
      FP    DB241.DBX   58.2;
      JNB   _009;
      L     1;
      T     DB240.DBW    4;
_009: NOP   0;
NETWORK
TITLE =공정 작업완료 RESET시 차종 요청 카운터 횟수 Clear
//db240.dbw6=차종 설정 요구 발생 횟수 저장 영역
      A(    ;
      A     #Work_Complete;
      FN    DB241.DBX   58.3;
      JNB   _00a;
      L     0;
      T     DB240.DBW    4;
      SET   ;
      SAVE  ;
      CLR   ;
_00a: A     BR;
      )     ;
      JNB   _00b;
      L     0;
      T     DB240.DBW    6;
_00b: NOP   0;
NETWORK
TITLE =공정 작업완료 SET시 log저장 함수 호출
//FC2=LOG 저장용 함수
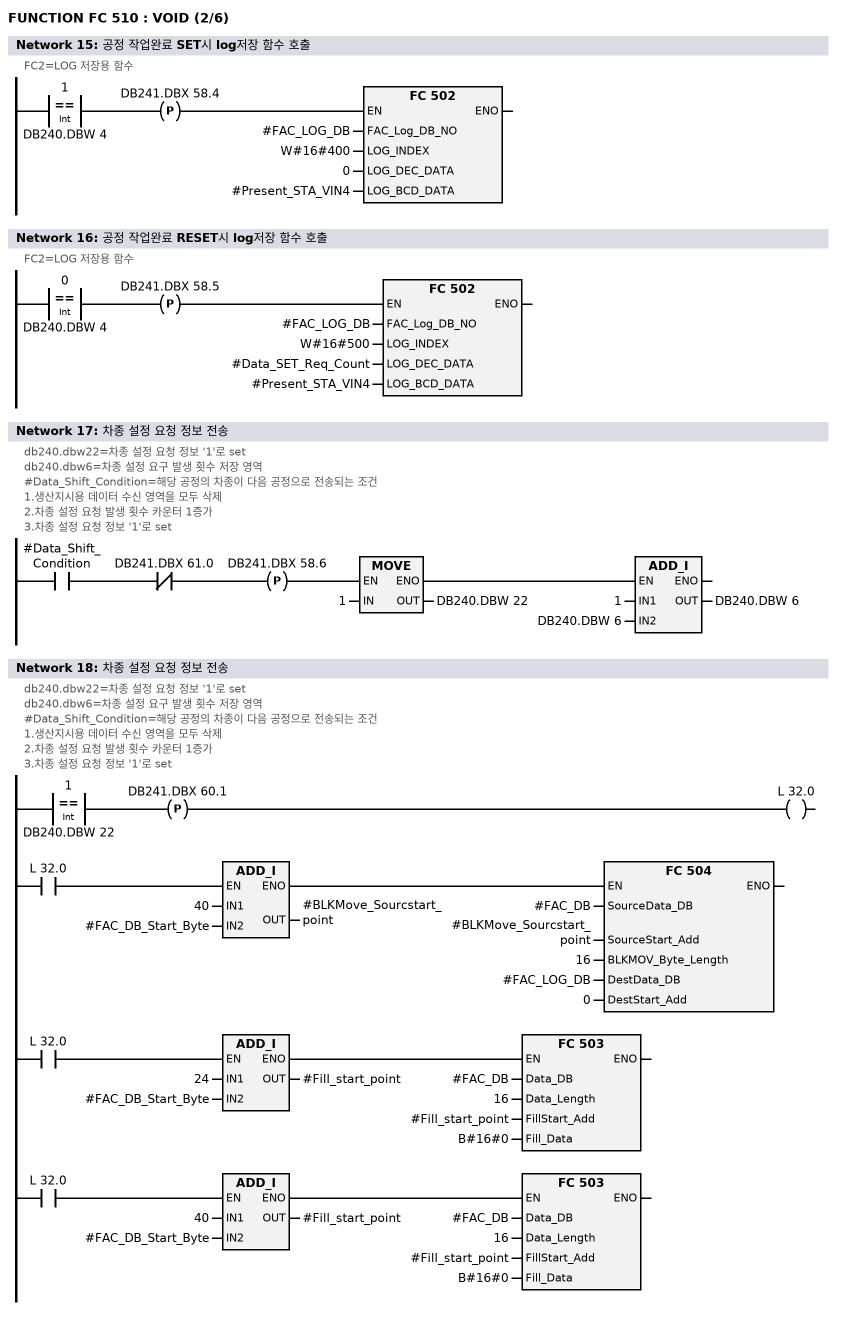
      A(    ;
      L     1;
      L     DB240.DBW    4;
      ==I   ;
      )     ;
      FP    DB241.DBX   58.4;
      JNB   _00c;
      CALL FC   502 (
           FAC_Log_DB_NO            := #FAC_LOG_DB,
           LOG_INDEX                := W#16#400,
           LOG_DEC_DATA             := 0,
           LOG_BCD_DATA             := #Present_STA_VIN4);
_00c: NOP   0;
NETWORK
TITLE =공정 작업완료 RESET시 log저장 함수 호출
//FC2=LOG 저장용 함수
      A(    ;
      L     0;
      L     DB240.DBW    4;
      ==I   ;
      )     ;
      FP    DB241.DBX   58.5;
      JNB   _00d;
      CALL FC   502 (
           FAC_Log_DB_NO            := #FAC_LOG_DB,
           LOG_INDEX                := W#16#500,
           LOG_DEC_DATA             := #Data_SET_Req_Count,
           LOG_BCD_DATA             := #Present_STA_VIN4);
_00d: NOP   0;
NETWORK
TITLE =차종 설정 요청 정보 전송
//db240.dbw22=차종 설정 요청 정보 '1'로 set
//db240.dbw6=차종 설정 요구 발생 횟수 저장 영역
//
//#Data_Shift_Condition=해당 공정의 차종이 다음 공정으로 전송되는 조건
//
//1.생산지시용 데이터 수신 영역을 모두 삭제
//2.차종 설정 요청 발생 횟수 카운터 1증가
//3.차종 설정 요청 정보 '1'로 set
      A(    ;
      A     #Data_Shift_Condition;
      AN    DB241.DBX   61.0;
      FP    DB241.DBX   58.6;
      JNB   _00e;
      L     1;
      T     DB240.DBW   22;
      SET   ;
      SAVE  ;
      CLR   ;
_00e: A     BR;
      )     ;
      JNB   _00f;
      L     1;
      L     DB240.DBW    6;
      +I    ;
      T     DB240.DBW    6;
_00f: NOP   0;
NETWORK
TITLE =차종 설정 요청 정보 전송
//db240.dbw22=차종 설정 요청 정보 '1'로 set
//db240.dbw6=차종 설정 요구 발생 횟수 저장 영역
//
//#Data_Shift_Condition=해당 공정의 차종이 다음 공정으로 전송되는 조건
//
//1.생산지시용 데이터 수신 영역을 모두 삭제
//2.차종 설정 요청 발생 횟수 카운터 1증가
//3.차종 설정 요청 정보 '1'로 set
      A(    ;
      L     1;
      L     DB240.DBW   22;
      ==I   ;
      )     ;
      FP    DB241.DBX   60.1;
      =     L     32.0;
      A(    ;
      A     L     32.0;
      JNB   _010;
      L     40;
      L     #FAC_DB_Start_Byte;
      +I    ;
      T     #BLKMove_Sourcstart_point;
      AN    OV;
      SAVE  ;
      CLR   ;
_010: A     BR;
      )     ;
      JNB   _011;
      CALL FC   504 (
           SourceData_DB            := #FAC_DB,
           SourceStart_Add          := #BLKMove_Sourcstart_point,
           BLKMOV_Byte_Length       := 16,
           DestData_DB              := #FAC_LOG_DB,
           DestStart_Add            := 0);
_011: NOP   0;
      A(    ;
      A     L     32.0;
      JNB   _012;
      L     24;
      L     #FAC_DB_Start_Byte;
      +I    ;
      T     #Fill_start_point;
      AN    OV;
      SAVE  ;
      CLR   ;
_012: A     BR;
      )     ;
      JNB   _013;
      CALL FC   503 (
           Data_DB                  := #FAC_DB,
           Data_Length              := 16,
           FillStart_Add            := #Fill_start_point,
           Fill_Data                := B#16#0);
_013: NOP   0;
      A(    ;
      A     L     32.0;
      JNB   _014;
      L     40;
      L     #FAC_DB_Start_Byte;
      +I    ;
      T     #Fill_start_point;
      AN    OV;
      SAVE  ;
      CLR   ;
_014: A     BR;
      )     ;
      JNB   _015;
      CALL FC   503 (
           Data_DB                  := #FAC_DB,
           Data_Length              := 16,
           FillStart_Add            := #Fill_start_point,
           Fill_Data                := B#16#0);
_015: NOP   0;
NETWORK
TITLE =차종 설정 요청 발생 횟수 정보를 Temp영역으로 전송
//db240.dbw6=차종 설정 요구 발생 횟수 저장 영역
//#Data_SET_Req_Count==차종 설정 요구 발생 횟수 임시(Log저장용) 저장 영역
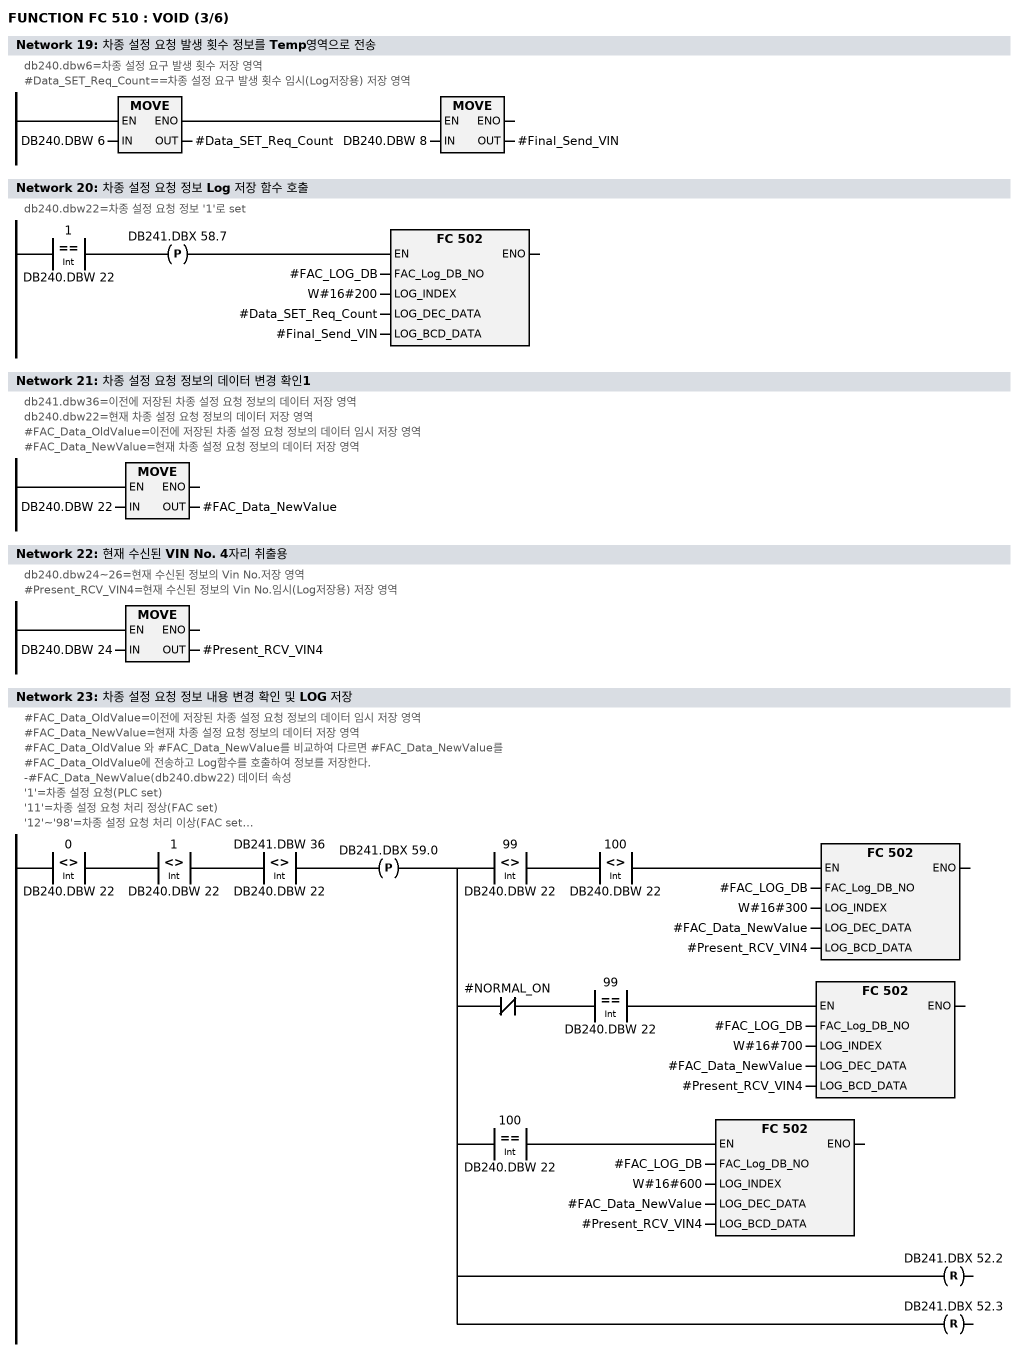
      A(    ;
      L     DB240.DBW    6;
      T     #Data_SET_Req_Count;
      SET   ;
      SAVE  ;
      CLR   ;
      A     BR;
      )     ;
      JNB   _016;
      L     DB240.DBW    8;
      T     #Final_Send_VIN;
_016: NOP   0;
NETWORK
TITLE =차종 설정 요청 정보 Log 저장 함수 호출
//db240.dbw22=차종 설정 요청 정보 '1'로 set
      A(    ;
      L     1;
      L     DB240.DBW   22;
      ==I   ;
      )     ;
      FP    DB241.DBX   58.7;
      JNB   _017;
      CALL FC   502 (
           FAC_Log_DB_NO            := #FAC_LOG_DB,
           LOG_INDEX                := W#16#200,
           LOG_DEC_DATA             := #Data_SET_Req_Count,
           LOG_BCD_DATA             := #Final_Send_VIN);
_017: NOP   0;
NETWORK
TITLE =차종 설정 요청 정보의 데이터 변경 확인1
//db241.dbw36=이전에 저장된 차종 설정 요청 정보의 데이터 저장 영역
//db240.dbw22=현재 차종 설정 요청 정보의 데이터 저장 영역
//#FAC_Data_OldValue=이전에 저장된 차종 설정 요청 정보의 데이터 임시 저장 영역
//#FAC_Data_NewValue=현재 차종 설정 요청 정보의 데이터 저장 영역
      L     DB240.DBW   22;
      T     #FAC_Data_NewValue;
      NOP   0;
NETWORK
TITLE =현재 수신된 VIN No. 4자리 취출용
//db240.dbw24~26=현재 수신된 정보의 Vin No.저장 영역
//#Present_RCV_VIN4=현재 수신된 정보의 Vin No.임시(Log저장용) 저장 영역
      L     DB240.DBW   24;
      T     #Present_RCV_VIN4;
      NOP   0;
NETWORK
TITLE =차종 설정 요청 정보 내용 변경 확인 및 LOG 저장
//#FAC_Data_OldValue=이전에 저장된 차종 설정 요청 정보의 데이터 임시 저장 영역
//#FAC_Data_NewValue=현재 차종 설정 요청 정보의 데이터 저장 영역
//#FAC_Data_OldValue 와 #FAC_Data_NewValue를 비교하여 다르면 #FAC_Data_NewValue를
//#FAC_Data_OldValue에 전송하고 Log함수를 호출하여 정보를 저장한다.
//
//-#FAC_Data_NewValue(db240.dbw22) 데이터 속성
//'1'=차종 설정 요청(PLC set)
//'11'=차종 설정 요청 처리 정상(FAC set)
//'12'~'98'=차종 설정 요청 처리 이상(FAC set)
//'99'=서열 데이터 부족(FAC set)
//'100'=차종 강제(수동) 설정(FAC set)
//db241.dbx54.7 pls삭제함
      A(    ;
      L     0;
      L     DB240.DBW   22;
      <>I   ;
      )     ;
      A(    ;
      L     1;
      L     DB240.DBW   22;
      <>I   ;
      )     ;
      A(    ;
      L     DB241.DBW   36;
      L     DB240.DBW   22;
      <>I   ;
      )     ;
      FP    DB241.DBX   59.0;
      =     L     32.0;
      A     L     32.0;
      A(    ;
      L     99;
      L     DB240.DBW   22;
      <>I   ;
      )     ;
      A(    ;
      L     100;
      L     DB240.DBW   22;
      <>I   ;
      )     ;
      JNB   _018;
      CALL FC   502 (
           FAC_Log_DB_NO            := #FAC_LOG_DB,
           LOG_INDEX                := W#16#300,
           LOG_DEC_DATA             := #FAC_Data_NewValue,
           LOG_BCD_DATA             := #Present_RCV_VIN4);
_018: NOP   0;
      A     L     32.0;
      AN    #NORMAL_ON;
      A(    ;
      L     99;
      L     DB240.DBW   22;
      ==I   ;
      )     ;
      JNB   _019;
      CALL FC   502 (
           FAC_Log_DB_NO            := #FAC_LOG_DB,
           LOG_INDEX                := W#16#700,
           LOG_DEC_DATA             := #FAC_Data_NewValue,
           LOG_BCD_DATA             := #Present_RCV_VIN4);
_019: NOP   0;
      A     L     32.0;
      A(    ;
      L     100;
      L     DB240.DBW   22;
      ==I   ;
      )     ;
      JNB   _01a;
      CALL FC   502 (
           FAC_Log_DB_NO            := #FAC_LOG_DB,
           LOG_INDEX                := W#16#600,
           LOG_DEC_DATA             := #FAC_Data_NewValue,
           LOG_BCD_DATA             := #Present_RCV_VIN4);
_01a: NOP   0;
      A     L     32.0;
      BLD   102;
      R     DB241.DBX   52.2;
      A     L     32.0;
      BLD   102;
      R     DB241.DBX   52.3;
NETWORK
TITLE =차종 강제 설정시 차종 설정 요청 카운터 및 수신 비교 정보 clear
//db240.dbw22=차종 설정 요청 정보 ('100'=강제(수동)설정)
//db240.dbw6=차종 설정 요구 발생 횟수 저장 영역
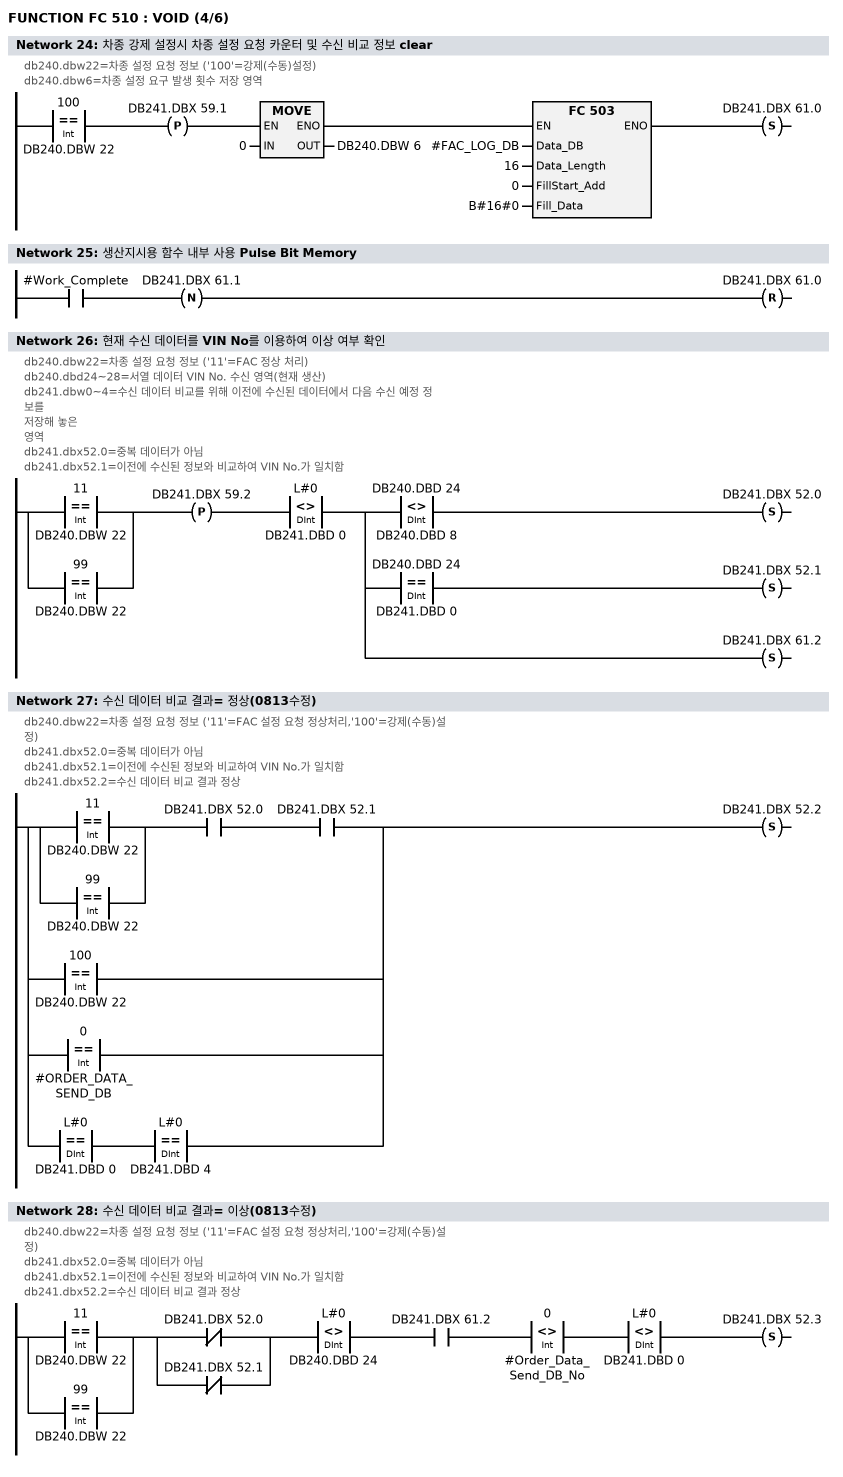
      A(    ;
      A(    ;
      L     100;
      L     DB240.DBW   22;
      ==I   ;
      )     ;
      FP    DB241.DBX   59.1;
      JNB   _01b;
      L     0;
      T     DB240.DBW    6;
      SET   ;
      SAVE  ;
      CLR   ;
_01b: A     BR;
      )     ;
      JNB   _01c;
      CALL FC   503 (
           Data_DB                  := #FAC_LOG_DB,
           Data_Length              := 16,
           FillStart_Add            := 0,
           Fill_Data                := B#16#0);
_01c: A     BR;
      S     DB241.DBX   61.0;
NETWORK
TITLE =생산지시용 함수 내부 사용 Pulse Bit Memory

      A     #Work_Complete;
      FN    DB241.DBX   61.1;
      R     DB241.DBX   61.0;
NETWORK
TITLE =현재 수신 데이터를 VIN No를 이용하여 이상 여부 확인
//db240.dbw22=차종 설정 요청 정보 ('11'=FAC 정상 처리)
//db240.dbd24~28=서열 데이터 VIN No. 수신 영역(현재 생산)
//db241.dbw0~4=수신 데이터 비교를 위해 이전에 수신된 데이터에서 다음 수신 예정 정
//보를
//저장해 놓은
//       영역
//db241.dbx52.0=중복 데이터가 아님
//db241.dbx52.1=이전에 수신된 정보와 비교하여 VIN No.가 일치함
      A(    ;
      O(    ;
      L     11;
      L     DB240.DBW   22;
      ==I   ;
      )     ;
      O(    ;
      L     99;
      L     DB240.DBW   22;
      ==I   ;
      )     ;
      )     ;
      FP    DB241.DBX   59.2;
      A(    ;
      L     L#0;
      L     DB241.DBD    0;
      <>D   ;
      )     ;
      =     L     32.0;
      A     L     32.0;
      A(    ;
      L     DB240.DBD   24;
      L     DB240.DBD    8;
      <>D   ;
      )     ;
      S     DB241.DBX   52.0;
      A     L     32.0;
      A(    ;
      L     DB240.DBD   24;
      L     DB241.DBD    0;
      ==D   ;
      )     ;
      S     DB241.DBX   52.1;
      A     L     32.0;
      BLD   102;
      S     DB241.DBX   61.2;
NETWORK
TITLE =수신 데이터 비교 결과= 정상(0813수정)
//db240.dbw22=차종 설정 요청 정보 ('11'=FAC 설정 요청 정상처리,'100'=강제(수동)설
//정)
//db241.dbx52.0=중복 데이터가 아님
//db241.dbx52.1=이전에 수신된 정보와 비교하여 VIN No.가 일치함
//db241.dbx52.2=수신 데이터 비교 결과 정상
      A(    ;
      O(    ;
      L     11;
      L     DB240.DBW   22;
      ==I   ;
      )     ;
      O(    ;
      L     99;
      L     DB240.DBW   22;
      ==I   ;
      )     ;
      )     ;
      A     DB241.DBX   52.0;
      A     DB241.DBX   52.1;
      O(    ;
      L     100;
      L     DB240.DBW   22;
      ==I   ;
      )     ;
      O(    ;
      L     0;
      L     #ORDER_DATA_SEND_DB;
      ==I   ;
      )     ;
      O     ;
      A(    ;
      L     L#0;
      L     DB241.DBD    0;
      ==D   ;
      )     ;
      A(    ;
      L     L#0;
      L     DB241.DBD    4;
      ==D   ;
      )     ;
      S     DB241.DBX   52.2;
NETWORK
TITLE =수신 데이터 비교 결과= 이상(0813수정)
//db240.dbw22=차종 설정 요청 정보 ('11'=FAC 설정 요청 정상처리,'100'=강제(수동)설
//정)
//db241.dbx52.0=중복 데이터가 아님
//db241.dbx52.1=이전에 수신된 정보와 비교하여 VIN No.가 일치함
//db241.dbx52.2=수신 데이터 비교 결과 정상
      A(    ;
      O(    ;
      L     11;
      L     DB240.DBW   22;
      ==I   ;
      )     ;
      O(    ;
      L     99;
      L     DB240.DBW   22;
      ==I   ;
      )     ;
      )     ;
      A(    ;
      ON    DB241.DBX   52.0;
      ON    DB241.DBX   52.1;
      )     ;
      A(    ;
      L     L#0;
      L     DB240.DBD   24;
      <>D   ;
      )     ;
      A     DB241.DBX   61.2;
      A(    ;
      L     0;
      L     #Order_Data_Send_DB_No;
      <>I   ;
      )     ;
      A(    ;
      L     L#0;
      L     DB241.DBD    0;
      <>D   ;
      )     ;
      S     DB241.DBX   52.3;
NETWORK
TITLE =서열 데이터 부족 출력 Set
//응답코드가 '99'일때 설비쪽으로 알려주기 위한 Logic
//응답코드 '99'=서열 데이터 부족
//db241.dbx52.3=서열 데이터 부족 Alarm 출력 보조
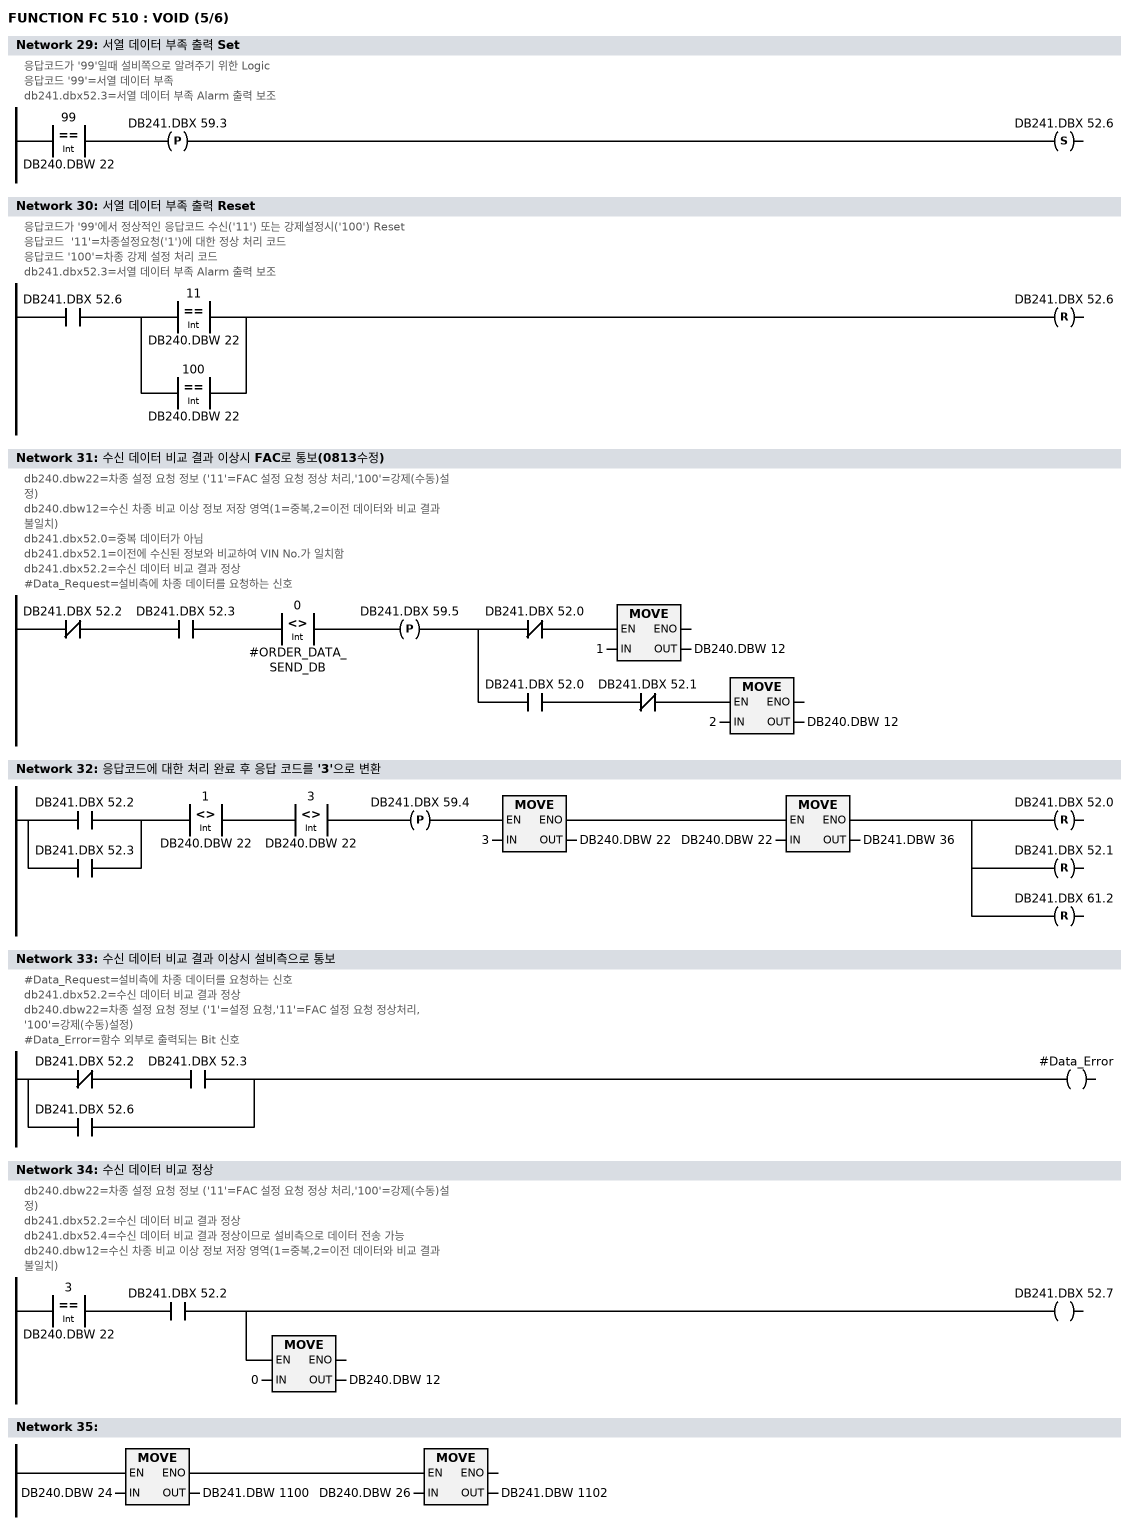
      A(    ;
      L     99;
      L     DB240.DBW   22;
      ==I   ;
      )     ;
      FP    DB241.DBX   59.3;
      S     DB241.DBX   52.6;
NETWORK
TITLE =서열 데이터 부족 출력 Reset
//응답코드가 '99'에서 정상적인 응답코드 수신('11') 또는 강제설정시('100') Reset
//응답코드  '11'=차종설정요청('1')에 대한 정상 처리 코드
//응답코드 '100'=차종 강제 설정 처리 코드
//db241.dbx52.3=서열 데이터 부족 Alarm 출력 보조
      A     DB241.DBX   52.6;
      A(    ;
      O(    ;
      L     11;
      L     DB240.DBW   22;
      ==I   ;
      )     ;
      O(    ;
      L     100;
      L     DB240.DBW   22;
      ==I   ;
      )     ;
      )     ;
      R     DB241.DBX   52.6;
NETWORK
TITLE =수신 데이터 비교 결과 이상시 FAC로 통보(0813수정)
//db240.dbw22=차종 설정 요청 정보 ('11'=FAC 설정 요청 정상 처리,'100'=강제(수동)설
//정)
//db240.dbw12=수신 차종 비교 이상 정보 저장 영역(1=중복,2=이전 데이터와 비교 결과
//불일치)
//db241.dbx52.0=중복 데이터가 아님
//db241.dbx52.1=이전에 수신된 정보와 비교하여 VIN No.가 일치함
//db241.dbx52.2=수신 데이터 비교 결과 정상
//#Data_Request=설비측에 차종 데이터를 요청하는 신호
      AN    DB241.DBX   52.2;
      A     DB241.DBX   52.3;
      A(    ;
      L     0;
      L     #ORDER_DATA_SEND_DB;
      <>I   ;
      )     ;
      FP    DB241.DBX   59.5;
      =     L     32.0;
      A     L     32.0;
      AN    DB241.DBX   52.0;
      JNB   _01d;
      L     1;
      T     DB240.DBW   12;
_01d: NOP   0;
      A     L     32.0;
      A     DB241.DBX   52.0;
      AN    DB241.DBX   52.1;
      JNB   _01e;
      L     2;
      T     DB240.DBW   12;
_01e: NOP   0;
NETWORK
TITLE =응답코드에 대한 처리 완료 후 응답 코드를 '3'으로 변환

      A(    ;
      A(    ;
      O     DB241.DBX   52.2;
      O     DB241.DBX   52.3;
      )     ;
      A(    ;
      L     1;
      L     DB240.DBW   22;
      <>I   ;
      )     ;
      A(    ;
      L     3;
      L     DB240.DBW   22;
      <>I   ;
      )     ;
      FP    DB241.DBX   59.4;
      JNB   _01f;
      L     3;
      T     DB240.DBW   22;
      SET   ;
      SAVE  ;
      CLR   ;
_01f: A     BR;
      )     ;
      JNB   _020;
      L     DB240.DBW   22;
      T     DB241.DBW   36;
      SET   ;
      SAVE  ;
      CLR   ;
_020: A     BR;
      R     DB241.DBX   52.0;
      R     DB241.DBX   52.1;
      R     DB241.DBX   61.2;
NETWORK
TITLE =수신 데이터 비교 결과 이상시 설비측으로 통보
//#Data_Request=설비측에 차종 데이터를 요청하는 신호
//db241.dbx52.2=수신 데이터 비교 결과 정상
//db240.dbw22=차종 설정 요청 정보 ('1'=설정 요청,'11'=FAC 설정 요청 정상처리,
//                         '100'=강제(수동)설정)
//#Data_Error=함수 외부로 출력되는 Bit 신호
      AN    DB241.DBX   52.2;
      A     DB241.DBX   52.3;
      O     DB241.DBX   52.6;
      =     #Data_Error;
NETWORK
TITLE =수신 데이터 비교 정상
//db240.dbw22=차종 설정 요청 정보 ('11'=FAC 설정 요청 정상 처리,'100'=강제(수동)설
//정)
//db241.dbx52.2=수신 데이터 비교 결과 정상
//db241.dbx52.4=수신 데이터 비교 결과 정상이므로 설비측으로 데이터 전송 가능
//db240.dbw12=수신 차종 비교 이상 정보 저장 영역(1=중복,2=이전 데이터와 비교 결과
//불일치)
      A(    ;
      L     3;
      L     DB240.DBW   22;
      ==I   ;
      )     ;
      A     DB241.DBX   52.2;
      =     L     32.0;
      A     L     32.0;
      BLD   102;
      =     DB241.DBX   52.7;
      A     L     32.0;
      JNB   _021;
      L     0;
      T     DB240.DBW   12;
_021: NOP   0;
NETWORK
TITLE =

      A(    ;
      L     DB240.DBW   24;
      T     DB241.DBW 1100;
      SET   ;
      SAVE  ;
      CLR   ;
      A     BR;
      )     ;
      JNB   _022;
      L     DB240.DBW   26;
      T     DB241.DBW 1102;
_022: NOP   0;
NETWORK
TITLE =
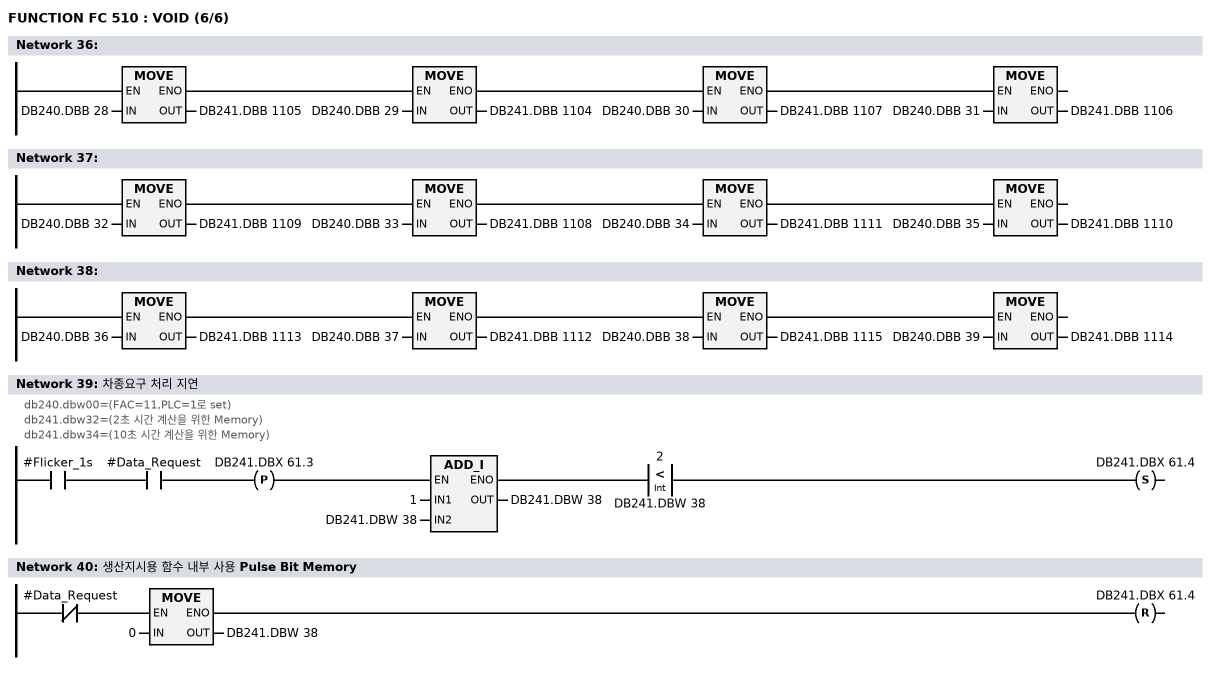

      A(    ;
      A(    ;
      A(    ;
      L     DB240.DBB   28;
      T     DB241.DBB 1105;
      SET   ;
      SAVE  ;
      CLR   ;
      A     BR;
      )     ;
      JNB   _023;
      L     DB240.DBB   29;
      T     DB241.DBB 1104;
      SET   ;
      SAVE  ;
      CLR   ;
_023: A     BR;
      )     ;
      JNB   _024;
      L     DB240.DBB   30;
      T     DB241.DBB 1107;
      SET   ;
      SAVE  ;
      CLR   ;
_024: A     BR;
      )     ;
      JNB   _025;
      L     DB240.DBB   31;
      T     DB241.DBB 1106;
_025: NOP   0;
NETWORK
TITLE =

      A(    ;
      A(    ;
      A(    ;
      L     DB240.DBB   32;
      T     DB241.DBB 1109;
      SET   ;
      SAVE  ;
      CLR   ;
      A     BR;
      )     ;
      JNB   _026;
      L     DB240.DBB   33;
      T     DB241.DBB 1108;
      SET   ;
      SAVE  ;
      CLR   ;
_026: A     BR;
      )     ;
      JNB   _027;
      L     DB240.DBB   34;
      T     DB241.DBB 1111;
      SET   ;
      SAVE  ;
      CLR   ;
_027: A     BR;
      )     ;
      JNB   _028;
      L     DB240.DBB   35;
      T     DB241.DBB 1110;
_028: NOP   0;
NETWORK
TITLE =

      A(    ;
      A(    ;
      A(    ;
      L     DB240.DBB   36;
      T     DB241.DBB 1113;
      SET   ;
      SAVE  ;
      CLR   ;
      A     BR;
      )     ;
      JNB   _029;
      L     DB240.DBB   37;
      T     DB241.DBB 1112;
      SET   ;
      SAVE  ;
      CLR   ;
_029: A     BR;
      )     ;
      JNB   _02a;
      L     DB240.DBB   38;
      T     DB241.DBB 1115;
      SET   ;
      SAVE  ;
      CLR   ;
_02a: A     BR;
      )     ;
      JNB   _02b;
      L     DB240.DBB   39;
      T     DB241.DBB 1114;
_02b: NOP   0;
NETWORK
TITLE =차종요구 처리 지연
//db240.dbw00=(FAC=11,PLC=1로 set)
//db241.dbw32=(2초 시간 계산을 위한 Memory)
//db241.dbw34=(10초 시간 계산을 위한 Memory)
      A(    ;
      A     #Flicker_1s;
      A     #Data_Request;
      FP    DB241.DBX   61.3;
      JNB   _02c;
      L     1;
      L     DB241.DBW   38;
      +I    ;
      T     DB241.DBW   38;
      AN    OV;
      SAVE  ;
      CLR   ;
_02c: A     BR;
      )     ;
      A(    ;
      L     2;
      L     DB241.DBW   38;
      <I    ;
      )     ;
      S     DB241.DBX   61.4;
NETWORK
TITLE =생산지시용 함수 내부 사용 Pulse Bit Memory

      AN    #Data_Request;
      JNB   _02d;
      L     0;
      T     DB241.DBW   38;
      SET   ;
      SAVE  ;
      CLR   ;
_02d: A     BR;
      R     DB241.DBX   61.4;
NETWORK
TITLE =설비측 차종 요청 ON시 데이터 전송
//db240.dbw22=생산지시 ON/OFF 선택 정보(1=ON)
//#Data_Request=함수로 입력된 신호(설비측에서 차종 데이터 요구)
//db241.dbx50.3=수신 데이터 비교 결과 정상이므로 설비측으로 데이터 전송 가능
//
//1.수신 데이터를 설비측으로 #Order_Data_Send_DB_No의
//#Order_Data_Send_DB_Byte부터
//  16Byte를 전송
//2.설비측으로 전송한 데이터에서 VIN No.(공정 최종 전송)를 DB에 저장
//3.다음에 수신할 데이터를 비교하기 위해 FAC Log저장용 DB에 전송
      A(    ;
      L     1;
      L     DB240.DBW    2;
      ==I   ;
      )     ;
      A(    ;
      L     3;
      L     DB240.DBW   22;
      ==I   ;
      )     ;
      A     #Data_Request;
      A     DB241.DBX   61.4;
      A     DB241.DBX   52.7;
      =     L     32.0;
      A     L     32.0;
      JNB   _02e;
      CALL FC   504 (
           SourceData_DB            := #FAC_LOG_DB,
           SourceStart_Add          := 1100,
           BLKMOV_Byte_Length       := 16,
           DestData_DB              := #Order_Data_Send_DB_No,
           DestStart_Add            := #Order_Data_Send_DB_Byte);
_02e: A     BR;
      R     DB241.DBX   61.0;
      A(    ;
      A(    ;
      A     L     32.0;
      JNB   _02f;
      L     24;
      L     #FAC_DB_Start_Byte;
      +I    ;
      T     #BLKMove_Sourcstart_point;
      AN    OV;
      SAVE  ;
      CLR   ;
_02f: A     BR;
      )     ;
      JNB   _030;
      L     8;
      L     #FAC_DB_Start_Byte;
      +I    ;
      T     #BLKMove_Deststart_point;
      AN    OV;
      SAVE  ;
      CLR   ;
_030: A     BR;
      )     ;
      JNB   _031;
      CALL FC   504 (
           SourceData_DB            := #FAC_DB,
           SourceStart_Add          := #BLKMove_Sourcstart_point,
           BLKMOV_Byte_Length       := 4,
           DestData_DB              := #FAC_DB,
           DestStart_Add            := #BLKMove_Deststart_point);
_031: NOP   0;
      A(    ;
      A     L     32.0;
      JNB   _032;
      L     40;
      L     #FAC_DB_Start_Byte;
      +I    ;
      T     #BLKMove_Sourcstart_point;
      AN    OV;
      SAVE  ;
      CLR   ;
_032: A     BR;
      )     ;
      JNB   _033;
      CALL FC   504 (
           SourceData_DB            := #FAC_DB,
           SourceStart_Add          := #BLKMove_Sourcstart_point,
           BLKMOV_Byte_Length       := 16,
           DestData_DB              := #FAC_LOG_DB,
           DestStart_Add            := 0);
_033: NOP   0;
NETWORK
TITLE = 현재 공정 차종 영역에서 운영 정보 bit확인
//db241.dbx26.2~7=차종 영역 표준Map에서 운영정보용 BIT
//db241.dbx54.0=차종 영역에 운영 정보 있음
//db241.dbx54.1=차종 영역에 운영 정보 있음 기억
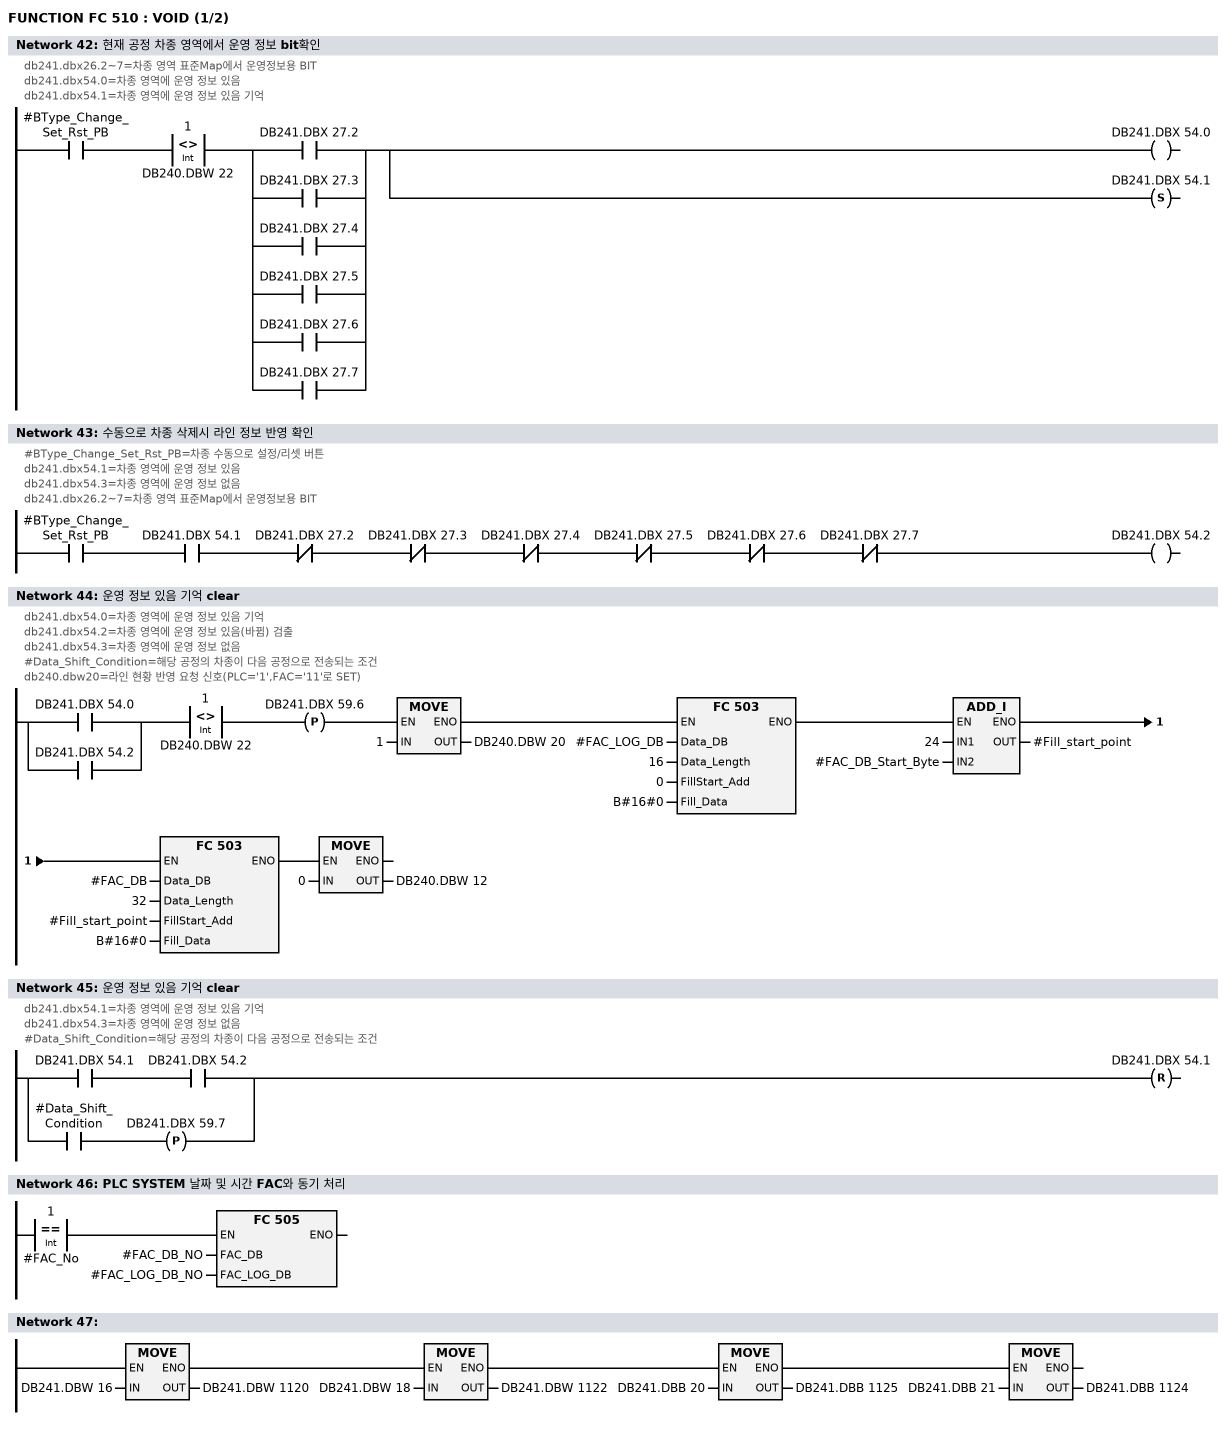
      A     #BType_Change_Set_Rst_PB;
      A(    ;
      L     1;
      L     DB240.DBW   22;
      <>I   ;
      )     ;
      A(    ;
      O     DB241.DBX   27.2;
      O     DB241.DBX   27.3;
      O     DB241.DBX   27.4;
      O     DB241.DBX   27.5;
      O     DB241.DBX   27.6;
      O     DB241.DBX   27.7;
      )     ;
      =     DB241.DBX   54.0;
      S     DB241.DBX   54.1;
NETWORK
TITLE =수동으로 차종 삭제시 라인 정보 반영 확인
//#BType_Change_Set_Rst_PB=차종 수동으로 설정/리셋 버튼
//db241.dbx54.1=차종 영역에 운영 정보 있음
//db241.dbx54.3=차종 영역에 운영 정보 없음
//db241.dbx26.2~7=차종 영역 표준Map에서 운영정보용 BIT
      A     #BType_Change_Set_Rst_PB;
      A     DB241.DBX   54.1;
      AN    DB241.DBX   27.2;
      AN    DB241.DBX   27.3;
      AN    DB241.DBX   27.4;
      AN    DB241.DBX   27.5;
      AN    DB241.DBX   27.6;
      AN    DB241.DBX   27.7;
      =     DB241.DBX   54.2;
NETWORK
TITLE =운영 정보 있음 기억 clear
//db241.dbx54.0=차종 영역에 운영 정보 있음 기억
//db241.dbx54.2=차종 영역에 운영 정보 있음(바뀜) 검출
//db241.dbx54.3=차종 영역에 운영 정보 없음
//#Data_Shift_Condition=해당 공정의 차종이 다음 공정으로 전송되는 조건
//db240.dbw20=라인 현황 반영 요청 신호(PLC='1',FAC='11'로 SET)
      A(    ;
      A(    ;
      A(    ;
      A(    ;
      A(    ;
      O     DB241.DBX   54.0;
      O     DB241.DBX   54.2;
      )     ;
      A(    ;
      L     1;
      L     DB240.DBW   22;
      <>I   ;
      )     ;
      FP    DB241.DBX   59.6;
      JNB   _034;
      L     1;
      T     DB240.DBW   20;
      SET   ;
      SAVE  ;
      CLR   ;
_034: A     BR;
      )     ;
      JNB   _035;
      CALL FC   503 (
           Data_DB                  := #FAC_LOG_DB,
           Data_Length              := 16,
           FillStart_Add            := 0,
           Fill_Data                := B#16#0);
_035: A     BR;
      )     ;
      JNB   _036;
      L     24;
      L     #FAC_DB_Start_Byte;
      +I    ;
      T     #Fill_start_point;
      AN    OV;
      SAVE  ;
      CLR   ;
_036: A     BR;
      )     ;
      JNB   _037;
      CALL FC   503 (
           Data_DB                  := #FAC_DB,
           Data_Length              := 32,
           FillStart_Add            := #Fill_start_point,
           Fill_Data                := B#16#0);
_037: A     BR;
      )     ;
      JNB   _038;
      L     0;
      T     DB240.DBW   12;
_038: NOP   0;
NETWORK
TITLE =운영 정보 있음 기억 clear
//db241.dbx54.1=차종 영역에 운영 정보 있음 기억
//db241.dbx54.3=차종 영역에 운영 정보 없음
//#Data_Shift_Condition=해당 공정의 차종이 다음 공정으로 전송되는 조건
      A     DB241.DBX   54.1;
      A     DB241.DBX   54.2;
      O(    ;
      A     #Data_Shift_Condition;
      FP    DB241.DBX   59.7;
      )     ;
      R     DB241.DBX   54.1;
NETWORK
TITLE =PLC SYSTEM 날짜 및 시간 FAC와 동기 처리

      A(    ;
      L     1;
      L     #FAC_No;
      ==I   ;
      )     ;
      JNB   _039;
      CALL FC   505 (
           FAC_DB                   := #FAC_DB_NO,
           FAC_LOG_DB               := #FAC_LOG_DB_NO);
_039: NOP   0;
NETWORK
TITLE =

      A(    ;
      A(    ;
      A(    ;
      L     DB241.DBW   16;
      T     DB241.DBW 1120;
      SET   ;
      SAVE  ;
      CLR   ;
      A     BR;
      )     ;
      JNB   _03a;
      L     DB241.DBW   18;
      T     DB241.DBW 1122;
      SET   ;
      SAVE  ;
      CLR   ;
_03a: A     BR;
      )     ;
      JNB   _03b;
      L     DB241.DBB   20;
      T     DB241.DBB 1125;
      SET   ;
      SAVE  ;
      CLR   ;
_03b: A     BR;
      )     ;
      JNB   _03c;
      L     DB241.DBB   21;
      T     DB241.DBB 1124;
_03c: NOP   0;
NETWORK
TITLE =
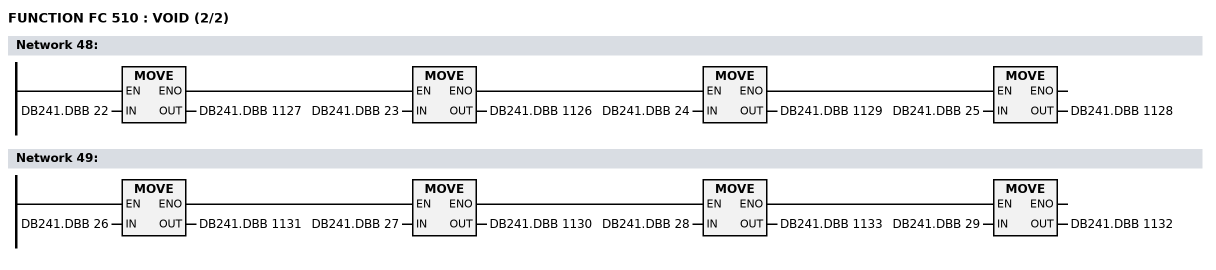

      A(    ;
      A(    ;
      A(    ;
      L     DB241.DBB   22;
      T     DB241.DBB 1127;
      SET   ;
      SAVE  ;
      CLR   ;
      A     BR;
      )     ;
      JNB   _03d;
      L     DB241.DBB   23;
      T     DB241.DBB 1126;
      SET   ;
      SAVE  ;
      CLR   ;
_03d: A     BR;
      )     ;
      JNB   _03e;
      L     DB241.DBB   24;
      T     DB241.DBB 1129;
      SET   ;
      SAVE  ;
      CLR   ;
_03e: A     BR;
      )     ;
      JNB   _03f;
      L     DB241.DBB   25;
      T     DB241.DBB 1128;
_03f: NOP   0;
NETWORK
TITLE =

      A(    ;
      A(    ;
      A(    ;
      L     DB241.DBB   26;
      T     DB241.DBB 1131;
      SET   ;
      SAVE  ;
      CLR   ;
      A     BR;
      )     ;
      JNB   _040;
      L     DB241.DBB   27;
      T     DB241.DBB 1130;
      SET   ;
      SAVE  ;
      CLR   ;
_040: A     BR;
      )     ;
      JNB   _041;
      L     DB241.DBB   28;
      T     DB241.DBB 1133;
      SET   ;
      SAVE  ;
      CLR   ;
_041: A     BR;
      )     ;
      JNB   _042;
      L     DB241.DBB   29;
      T     DB241.DBB 1132;
_042: NOP   0;
END_FUNCTION

DATA_BLOCK DB 71
TITLE =
AUTHOR : SIMATIC
FAMILY : CPU_300
VERSION : 0.0

 FB 12
BEGIN
   REQ := FALSE;
   R := FALSE;
   ID := W#16#0;
   R_ID := DW#16#0;
   DONE := FALSE;
   ERROR := FALSE;
   STATUS := W#16#0;
   LEN := W#16#0;
   FB_ZUSTAND := B#16#0;
   REQ_SAVE := FALSE;
   R_SAVE := FALSE;
   ID_SAVE := W#16#0;
   R_ID_SAVE := DW#16#0;
   LEN_SAVE := W#16#0;
   SD_1_SAVE0 := W#16#0;
   SD_1_SAVE2 := W#16#0;
   SD_1_SAVE4 := W#16#0;
   SD_1_SAVE6 := W#16#0;
   SD_1_SAVE8 := W#16#0;
   HS_REQ_BYTE.rii := FALSE;
   HS_REQ_BYTE.nva := FALSE;
   HS_REQ_BYTE.ofs := FALSE;
   HS_REQ_BYTE.dir := FALSE;
   HS_REQ_BYTE.res := FALSE;
   HS_REQ_BYTE.roc := FALSE;
   HS_REQ_BYTE.nls := FALSE;
   HS_REQ_BYTE.rlo := FALSE;
   HS_RESP_BYTE.aii := FALSE;
   HS_RESP_BYTE.sns := FALSE;
   HS_RESP_BYTE.sqc := FALSE;
   HS_RESP_BYTE.ads := FALSE;
   HS_RESP_BYTE.aoc := FALSE;
   HS_RESP_BYTE.rs1 := FALSE;
   HS_RESP_BYTE.cnr := FALSE;
   HS_RESP_BYTE.rs2 := FALSE;
   HS_RESP_DSNR := B#16#0;
   HS_RESP_OFFSET := W#16#0;
   SD_1_WORD0 := W#16#0;
   SD_1_COUNT := W#16#0;
   SD_1_DBNUMMER := W#16#0;
   SD_1_DWORD6 := DW#16#0;
   SD_1_TYP := B#16#0;
   SFC_PARAM.LEN := W#16#0;
   SFC_PARAM.DB_NUMMER := W#16#0;
   SFC_PARAM.START := DW#16#0;
   BUFFER[0] := W#16#0;
   BUFFER[1] := W#16#0;
   BUFFER[2] := W#16#0;
   BUFFER[3] := W#16#0;
   BUFFER[4] := W#16#0;
   BUFFER[5] := W#16#0;
   BUFFER[6] := W#16#0;
   BUFFER[7] := W#16#0;
   BUFFER[8] := W#16#0;
   BUFFER[9] := W#16#0;
   BUFFER[10] := W#16#0;
   BUFFER[11] := W#16#0;
   BUFFER[12] := W#16#0;
   BUFFER[13] := W#16#0;
   BUFFER[14] := W#16#0;
   BUFFER[15] := W#16#0;
   BUFFER[16] := W#16#0;
   BUFFER[17] := W#16#0;
   BUFFER[18] := W#16#0;
   BUFFER[19] := W#16#0;
   BUFFER[20] := W#16#0;
   BUFFER[21] := W#16#0;
   BUFFER[22] := W#16#0;
   BUFFER[23] := W#16#0;
   BUFFER[24] := W#16#0;
   BUFFER[25] := W#16#0;
   BUFFER[26] := W#16#0;
   BUFFER[27] := W#16#0;
   BUFFER[28] := W#16#0;
   BUFFER[29] := W#16#0;
   BUFFER[30] := W#16#0;
   BUFFER[31] := W#16#0;
   BUFFER[32] := W#16#0;
   BUFFER[33] := W#16#0;
   BUFFER[34] := W#16#0;
   BUFFER[35] := W#16#0;
   BUFFER[36] := W#16#0;
   BUFFER[37] := W#16#0;
   BUFFER[38] := W#16#0;
   BUFFER[39] := W#16#0;
   BUFFER[40] := W#16#0;
   BUFFER[41] := W#16#0;
   BUFFER[42] := W#16#0;
   BUFFER[43] := W#16#0;
   BUFFER[44] := W#16#0;
   BUFFER[45] := W#16#0;
   BUFFER[46] := W#16#0;
   BUFFER[47] := W#16#0;
   BUFFER[48] := W#16#0;
   BUFFER[49] := W#16#0;
   BUFFER[50] := W#16#0;
   BUFFER[51] := W#16#0;
   BUFFER[52] := W#16#0;
   BUFFER[53] := W#16#0;
   BUFFER[54] := W#16#0;
   BUFFER[55] := W#16#0;
   BUFFER[56] := W#16#0;
   BUFFER[57] := W#16#0;
   BUFFER[58] := W#16#0;
   BUFFER[59] := W#16#0;
   BUFFER[60] := W#16#0;
   BUFFER[61] := W#16#0;
   BUFFER[62] := W#16#0;
   BUFFER[63] := W#16#0;
   BUFFER[64] := W#16#0;
   BUFFER[65] := W#16#0;
   BUFFER[66] := W#16#0;
   BUFFER[67] := W#16#0;
   BUFFER[68] := W#16#0;
   BUFFER[69] := W#16#0;
   BUFFER[70] := W#16#0;
   BUFFER[71] := W#16#0;
   BUFFER[72] := W#16#0;
   BUFFER[73] := W#16#0;
   BUFFER[74] := W#16#0;
   BUFFER[75] := W#16#0;
   BUFFER[76] := W#16#0;
   BUFFER[77] := W#16#0;
   BUFFER[78] := W#16#0;
   BUFFER[79] := W#16#0;
   BUFFER[80] := W#16#0;
   BUFFER[81] := W#16#0;
   BUFFER[82] := W#16#0;
   BUFFER[83] := W#16#0;
   BUFFER[84] := W#16#0;
   BUFFER[85] := W#16#0;
   BUFFER[86] := W#16#0;
   BUFFER[87] := W#16#0;
   BUFFER[88] := W#16#0;
   BUFFER[89] := W#16#0;
   BUFFER[90] := W#16#0;
   BUFFER[91] := W#16#0;
   BUFFER[92] := W#16#0;
   BUFFER[93] := W#16#0;
   BUFFER[94] := W#16#0;
   BUFFER[95] := W#16#0;
   BUFFER[96] := W#16#0;
   BUFFER[97] := W#16#0;
   BUFFER[98] := W#16#0;
   BUFFER[99] := W#16#0;
   BUFFER[100] := W#16#0;
   BUFFER[101] := W#16#0;
   BUFFER[102] := W#16#0;
   BUFFER[103] := W#16#0;
   BUFFER[104] := W#16#0;
   BUFFER[105] := W#16#0;
   BUFFER[106] := W#16#0;
   BUFFER[107] := W#16#0;
   BUFFER[108] := W#16#0;
   BUFFER[109] := W#16#0;
   BUFFER[110] := W#16#0;
   BUFFER[111] := W#16#0;
   BUFFER[112] := W#16#0;
   BUFFER[113] := W#16#0;
   BUFFER[114] := W#16#0;
   BUFFER[115] := W#16#0;
   BUFFER[116] := W#16#0;
   BUFFER[117] := W#16#0;
   BUFFER[118] := W#16#0;
   BUFFER[119] := W#16#0;
   REASON_FOR_CLOSE := B#16#0;
   DS_NR := B#16#0;
   PARAM_OFFSET := B#16#0;
   MAX_PUFF_LEN_SAVE := W#16#0;
   TYP_BOOL := FALSE;
   KANAL_PROBLEM := FALSE;
   KOMM_PROBLEM := FALSE;
   SEND_STARTED := FALSE;
   RECV_STARTED := FALSE;
   RESET_REQUEST := FALSE;
   RESET_EXECUTED := FALSE;
   DS200_BUSY := FALSE;
   MAX_DATA_LEN := W#16#0;
   LADDR_PTR := DW#16#0;
   FC_DATA_LEN := W#16#0;
   LADDR := W#16#0;
   SLEEP := B#16#0;
   SLEEP_EXT := B#16#0;
   ID_CLOSE := W#16#0;
   FB_KENNUNG := B#16#F1;
   RESERVE := B#16#0;
   ZUSTAND_WEICHE := B#16#0;
   SFB_AUFRUF.REQ := FALSE;
   SFB_AUFRUF.R := FALSE;
   SFB_AUFRUF.ID := W#16#0;
   SFB_AUFRUF.R_ID := DW#16#0;
   SFB_AUFRUF.DONE := FALSE;
   SFB_AUFRUF.ERROR := FALSE;
   SFB_AUFRUF.STATUS := W#16#0;
   SFB_AUFRUF.LEN := W#16#0;
   SFB_AUFRUF.INDEX := W#16#0;
   ZUSTAND_WEICHE_1 := B#16#0;
END_DATA_BLOCK

DATA_BLOCK DB 72
TITLE =
AUTHOR : SIMATIC
FAMILY : CPU_300
VERSION : 0.0

